   A_3225_TSC01_AT.InMonL := FALSE;
   A_3225_TSC01_AT.InMonMid := FALSE;
   A_3225_TSC01_AT.InMonH := FALSE;
   A_3225_TSC01_AT.InMonHH := FALSE;
   A_3225_TSC01_AT.spare0205 := FALSE;
   A_3225_TSC01_AT.InpFaultAI := FALSE;
   A_3225_TSC01_AT.InpFaultDev := FALSE;
   A_3225_TSC01_AT.InHWStop := FALSE;
   A_3225_TSC01_AT.InDPFault := FALSE;
   A_3225_TSC01_AT.InDisable := FALSE;
   A_3225_TSC01_AT.CmdFaultReset := FALSE;
   A_3225_TSC01_AT.InLocal := FALSE;
   A_3225_TSC01_AT.spare0305 := FALSE;
   A_3225_TSC01_AT.InReport := FALSE;
   A_3225_TSC01_AT.spare0307 := FALSE;
   A_3225_TSC01_AT.OutLL := FALSE;
   A_3225_TSC01_AT.OutL := FALSE;
   A_3225_TSC01_AT.OutH := FALSE;
   A_3225_TSC01_AT.OutHH := FALSE;
   A_3225_TSC01_AT.OutOverflow := FALSE;
   A_3225_TSC01_AT.spare0405 := FALSE;
   A_3225_TSC01_AT.OutFaultAI := FALSE;
   A_3225_TSC01_AT.spare0407 := FALSE;
   A_3225_TSC01_AT.StLL := FALSE;
   A_3225_TSC01_AT.StL := FALSE;
   A_3225_TSC01_AT.StMid := FALSE;
   A_3225_TSC01_AT.StH := FALSE;
   A_3225_TSC01_AT.StHH := FALSE;
   A_3225_TSC01_AT.StFaultAI := FALSE;
   A_3225_TSC01_AT.OutWarning := FALSE;
   A_3225_TSC01_AT.OutFaulted := FALSE;
   A_3225_TSC01_AT.InpValue := 0;
   A_3225_TSC01_AT.OutValuePc := 0;
   A_3225_TSC01_AT.OutValueUnits := L#0;
   A_3225_TSC01_AT.Msg.WarningDoneLL := FALSE;
   A_3225_TSC01_AT.Msg.WarningDoneL := FALSE;
   A_3225_TSC01_AT.Msg.WarningDoneMid := FALSE;
   A_3225_TSC01_AT.Msg.WarningDoneH := FALSE;
   A_3225_TSC01_AT.Msg.WarningDoneHH := FALSE;
   A_3225_TSC01_AT.Msg.FaultDoneLL := FALSE;
   A_3225_TSC01_AT.Msg.FaultDoneL := FALSE;
   A_3225_TSC01_AT.Msg.FaultDoneMid := FALSE;
   A_3225_TSC01_AT.Msg.FaultDoneH := FALSE;
   A_3225_TSC01_AT.Msg.FaultDoneHH := FALSE;
   A_3225_TSC01_AT.Msg.FaultDoneDev := FALSE;
   A_3225_TSC01_AT.Msg.FaultDoneAI := FALSE;
   A_3225_TSC01_AT.OutAlarmNrLog := 0;
   A_3225_TSC01_AT.Par.ParObjectNo := 29713;
   A_3225_TSC01_AT.Par.ParMsgType := 7252;
   A_3225_TSC01_AT.Par.ParHornCode := 11;
   A_3225_TSC01_AT.Par.ParLogOff := FALSE;
   A_3225_TSC01_AT.Par.ParSpare0401 := FALSE;
   A_3225_TSC01_AT.Par.ParValueByUser := FALSE;
   A_3225_TSC01_AT.Par.ParLimitsPc := TRUE;
   A_3225_TSC01_AT.Par.ParWago := FALSE;
   A_3225_TSC01_AT.Par.ParNoHornByWarning := FALSE;
   A_3225_TSC01_AT.Par.ParWarningLL := FALSE;
   A_3225_TSC01_AT.Par.ParWarningL := FALSE;
   A_3225_TSC01_AT.Par.ParWarningMid := FALSE;
   A_3225_TSC01_AT.Par.ParWarningH := FALSE;
   A_3225_TSC01_AT.Par.ParWarningHH := FALSE;
   A_3225_TSC01_AT.Par.ParPreAlarmLL := FALSE;
   A_3225_TSC01_AT.Par.ParPreAlarmL := FALSE;
   A_3225_TSC01_AT.Par.ParPreAlarmMid := FALSE;
   A_3225_TSC01_AT.Par.ParPreAlarmH := FALSE;
   A_3225_TSC01_AT.Par.ParPreAlarmHH := FALSE;
   A_3225_TSC01_AT.Par.ParUnitsByZeroDigit := L#0;
   A_3225_TSC01_AT.Par.ParUnitsByMaxDigit := L#16384;
   A_3225_TSC01_AT.Par.ParUnitsBy100Pc := L#10000;
   A_3225_TSC01_AT.Par.ParLimitLL := L#-1;
   A_3225_TSC01_AT.Par.ParLimitL := L#0;
   A_3225_TSC01_AT.Par.ParLimitH := L#7000;
   A_3225_TSC01_AT.Par.ParLimitHH := L#8000;
   A_3225_TSC01_AT.Par.ParMonTimeLL := 0;
   A_3225_TSC01_AT.Par.ParMonTimeL := 0;
   A_3225_TSC01_AT.Par.ParMonTimeMid := 0;
   A_3225_TSC01_AT.Par.ParMonTimeH := 0;
   A_3225_TSC01_AT.Par.ParMonTimeHH := 0;
   A_3225_TSC01_AT.Par.ParDelayTimeDown := 10;
   A_3225_TSC01_AT.Par.ParDelayTimeUp := 10;
   A_3225_TSC01_AT.Par.ParDelayTime := 30;
   A_3225_TSC01_AT.Par.OutMonTimeLL := 0;
   A_3225_TSC01_AT.Par.OutMonTimeL := 0;
   A_3225_TSC01_AT.Par.OutMonTimeMid := 0;
   A_3225_TSC01_AT.Par.OutMonTimeH := 0;
   A_3225_TSC01_AT.Par.OutMonTimeHH := 0;
   A_3225_TSC01_AT.Par.OutDelayTimeDown := 0;
   A_3225_TSC01_AT.Par.OutDelayTimeUp := 0;
   A_3225_TSC01_AT.Par.OutDelayTime := 0;
   A_3225_TSC01_AT.Par.Spare66 := 0;
   A_3225_TSC01_COM.InValuePC := 0;
   A_3225_TSC01_COM.InEnableRev := FALSE;
   A_3225_TSC01_COM.InEnableFwd := FALSE;
   A_3225_TSC01_COM.CmdFaultReset := FALSE;
   A_3225_TSC01_COM.OutRunningRev := FALSE;
   A_3225_TSC01_COM.OutRunningFwd := FALSE;
   A_3225_TSC01_COM.OutFault := FALSE;
   A_3225_TSC01_COM.MotorStStopped := FALSE;
   A_3225_TSC01_COM.Spare := FALSE;
   A_3225_TSC01_COM.OutValuePC := 0;
   A_3225_TSC01_COM.Input.StateWord_1.STATE_WORD_BIT_8 := FALSE;
   A_3225_TSC01_COM.Input.StateWord_1.STATE_WORD_BIT_9 := FALSE;
   A_3225_TSC01_COM.Input.StateWord_1.STATE_WORD_BIT_10 := FALSE;
   A_3225_TSC01_COM.Input.StateWord_1.STATE_WORD_BIT_11 := FALSE;
   A_3225_TSC01_COM.Input.StateWord_1.STATE_WORD_BIT_12 := FALSE;
   A_3225_TSC01_COM.Input.StateWord_1.STATE_WORD_BIT_13 := FALSE;
   A_3225_TSC01_COM.Input.StateWord_1.STATE_WORD_BIT_14 := FALSE;
   A_3225_TSC01_COM.Input.StateWord_1.STATE_WORD_BIT_15 := FALSE;
   A_3225_TSC01_COM.Input.StateWord_1.ENDSTUFE_FREIGEGEBEN := FALSE;
   A_3225_TSC01_COM.Input.StateWord_1.BETRIEBSBEREIT := FALSE;
   A_3225_TSC01_COM.Input.StateWord_1.PA_DATEN_FREIGEGEBEN := FALSE;
   A_3225_TSC01_COM.Input.StateWord_1.AKTUELL_INTEGRATORSATZ := FALSE;
   A_3225_TSC01_COM.Input.StateWord_1.AKTUELL_PARAMETERSATZ := FALSE;
   A_3225_TSC01_COM.Input.StateWord_1.STOERUNG_WARNUNG := FALSE;
   A_3225_TSC01_COM.Input.StateWord_1.LS_RECHTS_AKTIV := FALSE;
   A_3225_TSC01_COM.Input.StateWord_1.LS_LINKS_AKTIV := FALSE;
   A_3225_TSC01_COM.Input.ActualValue01 := 0;
   A_3225_TSC01_COM.Input.ActualValue02 := 0;
   A_3225_TSC01_COM.Input.ActualValue03 := 0;
   A_3225_TSC01_COM.Input.ActualValue04 := 0;
   A_3225_TSC01_COM.Input.ActualValue05 := 0;
   A_3225_TSC01_COM.Output.ControlWord_1.CONTROL_WORD_BIT_8 := FALSE;
   A_3225_TSC01_COM.Output.ControlWord_1.CONTROL_WORD_BIT_9 := FALSE;
   A_3225_TSC01_COM.Output.ControlWord_1.CONTROL_WORD_BIT_10 := FALSE;
   A_3225_TSC01_COM.Output.ControlWord_1.CONTROL_WORD_BIT_11 := FALSE;
   A_3225_TSC01_COM.Output.ControlWord_1.CONTROL_WORD_BIT_12 := FALSE;
   A_3225_TSC01_COM.Output.ControlWord_1.CONTROL_WORD_BIT_13 := FALSE;
   A_3225_TSC01_COM.Output.ControlWord_1.CONTROL_WORD_BIT_14 := FALSE;
   A_3225_TSC01_COM.Output.ControlWord_1.CONTROL_WORD_BIT_15 := FALSE;
   A_3225_TSC01_COM.Output.ControlWord_1.REGLERSPERRE := FALSE;
   A_3225_TSC01_COM.Output.ControlWord_1.FREIGABE_SCHNELLSTOPP := FALSE;
   A_3225_TSC01_COM.Output.ControlWord_1.FREIGABE_HALT := FALSE;
   A_3225_TSC01_COM.Output.ControlWord_1.HALTEREGELUNG := FALSE;
   A_3225_TSC01_COM.Output.ControlWord_1.INTEGRATOR := FALSE;
   A_3225_TSC01_COM.Output.ControlWord_1.PARAMETERSATZ := FALSE;
   A_3225_TSC01_COM.Output.ControlWord_1.RESET := FALSE;
   A_3225_TSC01_COM.Output.ControlWord_1.RESERVE_BIT_7 := FALSE;
   A_3225_TSC01_COM.Output.SetpointValue01 := 0;
   A_3225_TSC01_COM.Output.SetpointValue02 := 0;
   A_3225_TSC01_COM.Output.SetpointValue03 := 0;
   A_3225_TSC01_COM.Output.SetpointValue04 := 0;
   A_3225_TSC01_COM.Output.SetpointValue05 := 0;
   A_3225_TSC01_COM.Par.spare1 := 0;
   A_3225_TSC01_COM.Par.spare2 := 0;
   A_3225_TSC01_COM.Par.spare3 := 0;
   A_3225_TSC01_COM.Par.ParMovidrive := TRUE;
   A_3225_TSC01_COM.Par.ParSinamics := FALSE;
   A_3225_TSC01_COM.Par.ParMicromaster := FALSE;
   A_3225_TSC01_COM.Par.ParABB := FALSE;
   A_3225_TSC01_COM.Par.ParNord := FALSE;
   A_3225_TSC01_COM.Par.ParDanfoss := FALSE;
   A_3225_TSC01_COM.Par.ParIOByteNo := 0;
   A_3226_KCU04AI1.StCode := 0;
   A_3226_KCU04AI1.InMonLL := FALSE;
   A_3226_KCU04AI1.InMonL := FALSE;
   A_3226_KCU04AI1.InMonMid := FALSE;
   A_3226_KCU04AI1.InMonH := FALSE;
   A_3226_KCU04AI1.InMonHH := FALSE;
   A_3226_KCU04AI1.spare0205 := FALSE;
   A_3226_KCU04AI1.InpFaultAI := FALSE;
   A_3226_KCU04AI1.InpFaultDev := FALSE;
   A_3226_KCU04AI1.InHWStop := FALSE;
   A_3226_KCU04AI1.InDPFault := FALSE;
   A_3226_KCU04AI1.InDisable := FALSE;
   A_3226_KCU04AI1.CmdFaultReset := FALSE;
   A_3226_KCU04AI1.InLocal := FALSE;
   A_3226_KCU04AI1.spare0305 := FALSE;
   A_3226_KCU04AI1.InReport := FALSE;
   A_3226_KCU04AI1.spare0307 := FALSE;
   A_3226_KCU04AI1.OutLL := FALSE;
   A_3226_KCU04AI1.OutL := FALSE;
   A_3226_KCU04AI1.OutH := FALSE;
   A_3226_KCU04AI1.OutHH := FALSE;
   A_3226_KCU04AI1.OutOverflow := FALSE;
   A_3226_KCU04AI1.spare0405 := FALSE;
   A_3226_KCU04AI1.OutFaultAI := FALSE;
   A_3226_KCU04AI1.spare0407 := FALSE;
   A_3226_KCU04AI1.StLL := FALSE;
   A_3226_KCU04AI1.StL := FALSE;
   A_3226_KCU04AI1.StMid := FALSE;
   A_3226_KCU04AI1.StH := FALSE;
   A_3226_KCU04AI1.StHH := FALSE;
   A_3226_KCU04AI1.StFaultAI := FALSE;
   A_3226_KCU04AI1.OutWarning := FALSE;
   A_3226_KCU04AI1.OutFaulted := FALSE;
   A_3226_KCU04AI1.InpValue := 0;
   A_3226_KCU04AI1.OutValuePc := 0;
   A_3226_KCU04AI1.OutValueUnits := L#0;
   A_3226_KCU04AI1.Msg.WarningDoneLL := FALSE;
   A_3226_KCU04AI1.Msg.WarningDoneL := FALSE;
   A_3226_KCU04AI1.Msg.WarningDoneMid := FALSE;
   A_3226_KCU04AI1.Msg.WarningDoneH := FALSE;
   A_3226_KCU04AI1.Msg.WarningDoneHH := FALSE;
   A_3226_KCU04AI1.Msg.FaultDoneLL := FALSE;
   A_3226_KCU04AI1.Msg.FaultDoneL := FALSE;
   A_3226_KCU04AI1.Msg.FaultDoneMid := FALSE;
   A_3226_KCU04AI1.Msg.FaultDoneH := FALSE;
   A_3226_KCU04AI1.Msg.FaultDoneHH := FALSE;
   A_3226_KCU04AI1.Msg.FaultDoneDev := FALSE;
   A_3226_KCU04AI1.Msg.FaultDoneAI := FALSE;
   A_3226_KCU04AI1.OutAlarmNrLog := 0;
   A_3226_KCU04AI1.Par.ParObjectNo := 29715;
   A_3226_KCU04AI1.Par.ParMsgType := 7252;
   A_3226_KCU04AI1.Par.ParHornCode := 11;
   A_3226_KCU04AI1.Par.ParLogOff := FALSE;
   A_3226_KCU04AI1.Par.ParSpare0401 := FALSE;
   A_3226_KCU04AI1.Par.ParValueByUser := FALSE;
   A_3226_KCU04AI1.Par.ParLimitsPc := TRUE;
   A_3226_KCU04AI1.Par.ParWago := FALSE;
   A_3226_KCU04AI1.Par.ParNoHornByWarning := FALSE;
   A_3226_KCU04AI1.Par.ParWarningLL := FALSE;
   A_3226_KCU04AI1.Par.ParWarningL := FALSE;
   A_3226_KCU04AI1.Par.ParWarningMid := FALSE;
   A_3226_KCU04AI1.Par.ParWarningH := TRUE;
   A_3226_KCU04AI1.Par.ParWarningHH := FALSE;
   A_3226_KCU04AI1.Par.ParPreAlarmLL := FALSE;
   A_3226_KCU04AI1.Par.ParPreAlarmL := FALSE;
   A_3226_KCU04AI1.Par.ParPreAlarmMid := FALSE;
   A_3226_KCU04AI1.Par.ParPreAlarmH := FALSE;
   A_3226_KCU04AI1.Par.ParPreAlarmHH := FALSE;
   A_3226_KCU04AI1.Par.ParUnitsByZeroDigit := L#0;
   A_3226_KCU04AI1.Par.ParUnitsByMaxDigit := L#2000;
   A_3226_KCU04AI1.Par.ParUnitsBy100Pc := L#10000;
   A_3226_KCU04AI1.Par.ParLimitLL := L#-1;
   A_3226_KCU04AI1.Par.ParLimitL := L#0;
   A_3226_KCU04AI1.Par.ParLimitH := L#3150;
   A_3226_KCU04AI1.Par.ParLimitHH := L#3550;
   A_3226_KCU04AI1.Par.ParMonTimeLL := 0;
   A_3226_KCU04AI1.Par.ParMonTimeL := 0;
   A_3226_KCU04AI1.Par.ParMonTimeMid := 0;
   A_3226_KCU04AI1.Par.ParMonTimeH := 600;
   A_3226_KCU04AI1.Par.ParMonTimeHH := 0;
   A_3226_KCU04AI1.Par.ParDelayTimeDown := 10;
   A_3226_KCU04AI1.Par.ParDelayTimeUp := 10;
   A_3226_KCU04AI1.Par.ParDelayTime := 30;
   A_3226_KCU04AI1.Par.OutMonTimeLL := 0;
   A_3226_KCU04AI1.Par.OutMonTimeL := 0;
   A_3226_KCU04AI1.Par.OutMonTimeMid := 0;
   A_3226_KCU04AI1.Par.OutMonTimeH := 0;
   A_3226_KCU04AI1.Par.OutMonTimeHH := 0;
   A_3226_KCU04AI1.Par.OutDelayTimeDown := 0;
   A_3226_KCU04AI1.Par.OutDelayTimeUp := 0;
   A_3226_KCU04AI1.Par.OutDelayTime := 0;
   A_3226_KCU04AI1.Par.Spare66 := 0;
   A_3226_KCU04AI2.StCode := 0;
   A_3226_KCU04AI2.InMonLL := FALSE;
   A_3226_KCU04AI2.InMonL := FALSE;
   A_3226_KCU04AI2.InMonMid := FALSE;
   A_3226_KCU04AI2.InMonH := FALSE;
   A_3226_KCU04AI2.InMonHH := FALSE;
   A_3226_KCU04AI2.spare0205 := FALSE;
   A_3226_KCU04AI2.InpFaultAI := FALSE;
   A_3226_KCU04AI2.InpFaultDev := FALSE;
   A_3226_KCU04AI2.InHWStop := FALSE;
   A_3226_KCU04AI2.InDPFault := FALSE;
   A_3226_KCU04AI2.InDisable := FALSE;
   A_3226_KCU04AI2.CmdFaultReset := FALSE;
   A_3226_KCU04AI2.InLocal := FALSE;
   A_3226_KCU04AI2.spare0305 := FALSE;
   A_3226_KCU04AI2.InReport := FALSE;
   A_3226_KCU04AI2.spare0307 := FALSE;
   A_3226_KCU04AI2.OutLL := FALSE;
   A_3226_KCU04AI2.OutL := FALSE;
   A_3226_KCU04AI2.OutH := FALSE;
   A_3226_KCU04AI2.OutHH := FALSE;
   A_3226_KCU04AI2.OutOverflow := FALSE;
   A_3226_KCU04AI2.spare0405 := FALSE;
   A_3226_KCU04AI2.OutFaultAI := FALSE;
   A_3226_KCU04AI2.spare0407 := FALSE;
   A_3226_KCU04AI2.StLL := FALSE;
   A_3226_KCU04AI2.StL := FALSE;
   A_3226_KCU04AI2.StMid := FALSE;
   A_3226_KCU04AI2.StH := FALSE;
   A_3226_KCU04AI2.StHH := FALSE;
   A_3226_KCU04AI2.StFaultAI := FALSE;
   A_3226_KCU04AI2.OutWarning := FALSE;
   A_3226_KCU04AI2.OutFaulted := FALSE;
   A_3226_KCU04AI2.InpValue := 0;
   A_3226_KCU04AI2.OutValuePc := 0;
   A_3226_KCU04AI2.OutValueUnits := L#0;
   A_3226_KCU04AI2.Msg.WarningDoneLL := FALSE;
   A_3226_KCU04AI2.Msg.WarningDoneL := FALSE;
   A_3226_KCU04AI2.Msg.WarningDoneMid := FALSE;
   A_3226_KCU04AI2.Msg.WarningDoneH := FALSE;
   A_3226_KCU04AI2.Msg.WarningDoneHH := FALSE;
   A_3226_KCU04AI2.Msg.FaultDoneLL := FALSE;
   A_3226_KCU04AI2.Msg.FaultDoneL := FALSE;
   A_3226_KCU04AI2.Msg.FaultDoneMid := FALSE;
   A_3226_KCU04AI2.Msg.FaultDoneH := FALSE;
   A_3226_KCU04AI2.Msg.FaultDoneHH := FALSE;
   A_3226_KCU04AI2.Msg.FaultDoneDev := FALSE;
   A_3226_KCU04AI2.Msg.FaultDoneAI := FALSE;
   A_3226_KCU04AI2.OutAlarmNrLog := 0;
   A_3226_KCU04AI2.Par.ParObjectNo := 29716;
   A_3226_KCU04AI2.Par.ParMsgType := 7252;
   A_3226_KCU04AI2.Par.ParHornCode := 11;
   A_3226_KCU04AI2.Par.ParLogOff := FALSE;
   A_3226_KCU04AI2.Par.ParSpare0401 := FALSE;
   A_3226_KCU04AI2.Par.ParValueByUser := FALSE;
   A_3226_KCU04AI2.Par.ParLimitsPc := TRUE;
   A_3226_KCU04AI2.Par.ParWago := FALSE;
   A_3226_KCU04AI2.Par.ParNoHornByWarning := FALSE;
   A_3226_KCU04AI2.Par.ParWarningLL := FALSE;
   A_3226_KCU04AI2.Par.ParWarningL := FALSE;
   A_3226_KCU04AI2.Par.ParWarningMid := FALSE;
   A_3226_KCU04AI2.Par.ParWarningH := TRUE;
   A_3226_KCU04AI2.Par.ParWarningHH := FALSE;
   A_3226_KCU04AI2.Par.ParPreAlarmLL := FALSE;
   A_3226_KCU04AI2.Par.ParPreAlarmL := FALSE;
   A_3226_KCU04AI2.Par.ParPreAlarmMid := FALSE;
   A_3226_KCU04AI2.Par.ParPreAlarmH := FALSE;
   A_3226_KCU04AI2.Par.ParPreAlarmHH := FALSE;
   A_3226_KCU04AI2.Par.ParUnitsByZeroDigit := L#0;
   A_3226_KCU04AI2.Par.ParUnitsByMaxDigit := L#2000;
   A_3226_KCU04AI2.Par.ParUnitsBy100Pc := L#10000;
   A_3226_KCU04AI2.Par.ParLimitLL := L#-1;
   A_3226_KCU04AI2.Par.ParLimitL := L#0;
   A_3226_KCU04AI2.Par.ParLimitH := L#3150;
   A_3226_KCU04AI2.Par.ParLimitHH := L#3550;
   A_3226_KCU04AI2.Par.ParMonTimeLL := 0;
   A_3226_KCU04AI2.Par.ParMonTimeL := 0;
   A_3226_KCU04AI2.Par.ParMonTimeMid := 0;
   A_3226_KCU04AI2.Par.ParMonTimeH := 600;
   A_3226_KCU04AI2.Par.ParMonTimeHH := 0;
   A_3226_KCU04AI2.Par.ParDelayTimeDown := 10;
   A_3226_KCU04AI2.Par.ParDelayTimeUp := 10;
   A_3226_KCU04AI2.Par.ParDelayTime := 30;
   A_3226_KCU04AI2.Par.OutMonTimeLL := 0;
   A_3226_KCU04AI2.Par.OutMonTimeL := 0;
   A_3226_KCU04AI2.Par.OutMonTimeMid := 0;
   A_3226_KCU04AI2.Par.OutMonTimeH := 0;
   A_3226_KCU04AI2.Par.OutMonTimeHH := 0;
   A_3226_KCU04AI2.Par.OutDelayTimeDown := 0;
   A_3226_KCU04AI2.Par.OutDelayTimeUp := 0;
   A_3226_KCU04AI2.Par.OutDelayTime := 0;
   A_3226_KCU04AI2.Par.Spare66 := 0;
   A_3226_BTE05.StCode := 0;
   A_3226_BTE05.InMonLL := FALSE;
   A_3226_BTE05.InMonL := FALSE;
   A_3226_BTE05.InMonMid := FALSE;
   A_3226_BTE05.InMonH := FALSE;
   A_3226_BTE05.InMonHH := FALSE;
   A_3226_BTE05.spare0205 := FALSE;
   A_3226_BTE05.InpFaultAI := FALSE;
   A_3226_BTE05.InpFaultDev := FALSE;
   A_3226_BTE05.InHWStop := FALSE;
   A_3226_BTE05.InDPFault := FALSE;
   A_3226_BTE05.InDisable := FALSE;
   A_3226_BTE05.CmdFaultReset := FALSE;
   A_3226_BTE05.InLocal := FALSE;
   A_3226_BTE05.spare0305 := FALSE;
   A_3226_BTE05.InReport := FALSE;
   A_3226_BTE05.spare0307 := FALSE;
   A_3226_BTE05.OutLL := FALSE;
   A_3226_BTE05.OutL := FALSE;
   A_3226_BTE05.OutH := FALSE;
   A_3226_BTE05.OutHH := FALSE;
   A_3226_BTE05.OutOverflow := FALSE;
   A_3226_BTE05.spare0405 := FALSE;
   A_3226_BTE05.OutFaultAI := FALSE;
   A_3226_BTE05.spare0407 := FALSE;
   A_3226_BTE05.StLL := FALSE;
   A_3226_BTE05.StL := FALSE;
   A_3226_BTE05.StMid := FALSE;
   A_3226_BTE05.StH := FALSE;
   A_3226_BTE05.StHH := FALSE;
   A_3226_BTE05.StFaultAI := FALSE;
   A_3226_BTE05.OutWarning := FALSE;
   A_3226_BTE05.OutFaulted := FALSE;
   A_3226_BTE05.InpValue := 0;
   A_3226_BTE05.OutValuePc := 0;
   A_3226_BTE05.OutValueUnits := L#0;
   A_3226_BTE05.Msg.WarningDoneLL := FALSE;
   A_3226_BTE05.Msg.WarningDoneL := FALSE;
   A_3226_BTE05.Msg.WarningDoneMid := FALSE;
   A_3226_BTE05.Msg.WarningDoneH := FALSE;
   A_3226_BTE05.Msg.WarningDoneHH := FALSE;
   A_3226_BTE05.Msg.FaultDoneLL := FALSE;
   A_3226_BTE05.Msg.FaultDoneL := FALSE;
   A_3226_BTE05.Msg.FaultDoneMid := FALSE;
   A_3226_BTE05.Msg.FaultDoneH := FALSE;
   A_3226_BTE05.Msg.FaultDoneHH := FALSE;
   A_3226_BTE05.Msg.FaultDoneDev := FALSE;
   A_3226_BTE05.Msg.FaultDoneAI := FALSE;
   A_3226_BTE05.OutAlarmNrLog := 0;
   A_3226_BTE05.Par.ParObjectNo := 29717;
   A_3226_BTE05.Par.ParMsgType := 7252;
   A_3226_BTE05.Par.ParHornCode := 11;
   A_3226_BTE05.Par.ParLogOff := FALSE;
   A_3226_BTE05.Par.ParSpare0401 := FALSE;
   A_3226_BTE05.Par.ParValueByUser := FALSE;
   A_3226_BTE05.Par.ParLimitsPc := TRUE;
   A_3226_BTE05.Par.ParWago := FALSE;
   A_3226_BTE05.Par.ParNoHornByWarning := FALSE;
   A_3226_BTE05.Par.ParWarningLL := FALSE;
   A_3226_BTE05.Par.ParWarningL := FALSE;
   A_3226_BTE05.Par.ParWarningMid := FALSE;
   A_3226_BTE05.Par.ParWarningH := TRUE;
   A_3226_BTE05.Par.ParWarningHH := FALSE;
   A_3226_BTE05.Par.ParPreAlarmLL := FALSE;
   A_3226_BTE05.Par.ParPreAlarmL := FALSE;
   A_3226_BTE05.Par.ParPreAlarmMid := FALSE;
   A_3226_BTE05.Par.ParPreAlarmH := FALSE;
   A_3226_BTE05.Par.ParPreAlarmHH := FALSE;
   A_3226_BTE05.Par.ParUnitsByZeroDigit := L#0;
   A_3226_BTE05.Par.ParUnitsByMaxDigit := L#27384;
   A_3226_BTE05.Par.ParUnitsBy100Pc := L#10000;
   A_3226_BTE05.Par.ParLimitLL := L#0;
   A_3226_BTE05.Par.ParLimitL := L#2000;
   A_3226_BTE05.Par.ParLimitH := L#8000;
   A_3226_BTE05.Par.ParLimitHH := L#10000;
   A_3226_BTE05.Par.ParMonTimeLL := 0;
   A_3226_BTE05.Par.ParMonTimeL := 0;
   A_3226_BTE05.Par.ParMonTimeMid := 0;
   A_3226_BTE05.Par.ParMonTimeH := 600;
   A_3226_BTE05.Par.ParMonTimeHH := 0;
   A_3226_BTE05.Par.ParDelayTimeDown := 10;
   A_3226_BTE05.Par.ParDelayTimeUp := 10;
   A_3226_BTE05.Par.ParDelayTime := 30;
   A_3226_BTE05.Par.OutMonTimeLL := 0;
   A_3226_BTE05.Par.OutMonTimeL := 0;
   A_3226_BTE05.Par.OutMonTimeMid := 0;
   A_3226_BTE05.Par.OutMonTimeH := 0;
   A_3226_BTE05.Par.OutMonTimeHH := 0;
   A_3226_BTE05.Par.OutDelayTimeDown := 0;
   A_3226_BTE05.Par.OutDelayTimeUp := 0;
   A_3226_BTE05.Par.OutDelayTime := 0;
   A_3226_BTE05.Par.Spare66 := 0;
   A_3226_BTE06.StCode := 0;
   A_3226_BTE06.InMonLL := FALSE;
   A_3226_BTE06.InMonL := FALSE;
   A_3226_BTE06.InMonMid := FALSE;
   A_3226_BTE06.InMonH := FALSE;
   A_3226_BTE06.InMonHH := FALSE;
   A_3226_BTE06.spare0205 := FALSE;
   A_3226_BTE06.InpFaultAI := FALSE;
   A_3226_BTE06.InpFaultDev := FALSE;
   A_3226_BTE06.InHWStop := FALSE;
   A_3226_BTE06.InDPFault := FALSE;
   A_3226_BTE06.InDisable := FALSE;
   A_3226_BTE06.CmdFaultReset := FALSE;
   A_3226_BTE06.InLocal := FALSE;
   A_3226_BTE06.spare0305 := FALSE;
   A_3226_BTE06.InReport := FALSE;
   A_3226_BTE06.spare0307 := FALSE;
   A_3226_BTE06.OutLL := FALSE;
   A_3226_BTE06.OutL := FALSE;
   A_3226_BTE06.OutH := FALSE;
   A_3226_BTE06.OutHH := FALSE;
   A_3226_BTE06.OutOverflow := FALSE;
   A_3226_BTE06.spare0405 := FALSE;
   A_3226_BTE06.OutFaultAI := FALSE;
   A_3226_BTE06.spare0407 := FALSE;
   A_3226_BTE06.StLL := FALSE;
   A_3226_BTE06.StL := FALSE;
   A_3226_BTE06.StMid := FALSE;
   A_3226_BTE06.StH := FALSE;
   A_3226_BTE06.StHH := FALSE;
   A_3226_BTE06.StFaultAI := FALSE;
   A_3226_BTE06.OutWarning := FALSE;
   A_3226_BTE06.OutFaulted := FALSE;
   A_3226_BTE06.InpValue := 0;
   A_3226_BTE06.OutValuePc := 0;
   A_3226_BTE06.OutValueUnits := L#0;
   A_3226_BTE06.Msg.WarningDoneLL := FALSE;
   A_3226_BTE06.Msg.WarningDoneL := FALSE;
   A_3226_BTE06.Msg.WarningDoneMid := FALSE;
   A_3226_BTE06.Msg.WarningDoneH := FALSE;
   A_3226_BTE06.Msg.WarningDoneHH := FALSE;
   A_3226_BTE06.Msg.FaultDoneLL := FALSE;
   A_3226_BTE06.Msg.FaultDoneL := FALSE;
   A_3226_BTE06.Msg.FaultDoneMid := FALSE;
   A_3226_BTE06.Msg.FaultDoneH := FALSE;
   A_3226_BTE06.Msg.FaultDoneHH := FALSE;
   A_3226_BTE06.Msg.FaultDoneDev := FALSE;
   A_3226_BTE06.Msg.FaultDoneAI := FALSE;
   A_3226_BTE06.OutAlarmNrLog := 0;
   A_3226_BTE06.Par.ParObjectNo := 29718;
   A_3226_BTE06.Par.ParMsgType := 7252;
   A_3226_BTE06.Par.ParHornCode := 11;
   A_3226_BTE06.Par.ParLogOff := FALSE;
   A_3226_BTE06.Par.ParSpare0401 := FALSE;
   A_3226_BTE06.Par.ParValueByUser := FALSE;
   A_3226_BTE06.Par.ParLimitsPc := TRUE;
   A_3226_BTE06.Par.ParWago := FALSE;
   A_3226_BTE06.Par.ParNoHornByWarning := FALSE;
   A_3226_BTE06.Par.ParWarningLL := FALSE;
   A_3226_BTE06.Par.ParWarningL := FALSE;
   A_3226_BTE06.Par.ParWarningMid := FALSE;
   A_3226_BTE06.Par.ParWarningH := TRUE;
   A_3226_BTE06.Par.ParWarningHH := FALSE;
   A_3226_BTE06.Par.ParPreAlarmLL := FALSE;
   A_3226_BTE06.Par.ParPreAlarmL := FALSE;
   A_3226_BTE06.Par.ParPreAlarmMid := FALSE;
   A_3226_BTE06.Par.ParPreAlarmH := FALSE;
   A_3226_BTE06.Par.ParPreAlarmHH := FALSE;
   A_3226_BTE06.Par.ParUnitsByZeroDigit := L#0;
   A_3226_BTE06.Par.ParUnitsByMaxDigit := L#27384;
   A_3226_BTE06.Par.ParUnitsBy100Pc := L#10000;
   A_3226_BTE06.Par.ParLimitLL := L#0;
   A_3226_BTE06.Par.ParLimitL := L#2000;
   A_3226_BTE06.Par.ParLimitH := L#8000;
   A_3226_BTE06.Par.ParLimitHH := L#10000;
   A_3226_BTE06.Par.ParMonTimeLL := 0;
   A_3226_BTE06.Par.ParMonTimeL := 0;
   A_3226_BTE06.Par.ParMonTimeMid := 0;
   A_3226_BTE06.Par.ParMonTimeH := 600;
   A_3226_BTE06.Par.ParMonTimeHH := 0;
   A_3226_BTE06.Par.ParDelayTimeDown := 10;
   A_3226_BTE06.Par.ParDelayTimeUp := 10;
   A_3226_BTE06.Par.ParDelayTime := 30;
   A_3226_BTE06.Par.OutMonTimeLL := 0;
   A_3226_BTE06.Par.OutMonTimeL := 0;
   A_3226_BTE06.Par.OutMonTimeMid := 0;
   A_3226_BTE06.Par.OutMonTimeH := 0;
   A_3226_BTE06.Par.OutMonTimeHH := 0;
   A_3226_BTE06.Par.OutDelayTimeDown := 0;
   A_3226_BTE06.Par.OutDelayTimeUp := 0;
   A_3226_BTE06.Par.OutDelayTime := 0;
   A_3226_BTE06.Par.Spare66 := 0;
   A_3226_MXZ01MA.Ma.StCode := 0;
   A_3226_MXZ01MA.Ma.InEnableRev := FALSE;
   A_3226_MXZ01MA.Ma.InEnableFwd := FALSE;
   A_3226_MXZ01MA.Ma.InOverrideHLOutlet := FALSE;
   A_3226_MXZ01MA.Ma.spare0203 := FALSE;
   A_3226_MXZ01MA.Ma.OutEdgeFaultReset := FALSE;
   A_3226_MXZ01MA.Ma.OutFaultResetFcttst := FALSE;
   A_3226_MXZ01MA.Ma.InpControlEBM := FALSE;
   A_3226_MXZ01MA.Ma.InpLocked := FALSE;
   A_3226_MXZ01MA.Ma.CmdOff := FALSE;
   A_3226_MXZ01MA.Ma.CmdOn := FALSE;
   A_3226_MXZ01MA.Ma.CmdNext := FALSE;
   A_3226_MXZ01MA.Ma.CmdFaultReset := FALSE;
   A_3226_MXZ01MA.Ma.InLocal := FALSE;
   A_3226_MXZ01MA.Ma.InManual := FALSE;
   A_3226_MXZ01MA.Ma.CmdTestEBM := FALSE;
   A_3226_MXZ01MA.Ma.InSeqStop := FALSE;
   A_3226_MXZ01MA.Ma.OutWarning := FALSE;
   A_3226_MXZ01MA.Ma.InfBMTopOk := FALSE;
   A_3226_MXZ01MA.Ma.InfBMBottomOk := FALSE;
   A_3226_MXZ01MA.Ma.InfSMOk := FALSE;
   A_3226_MXZ01MA.Ma.OutpFcttst_BM_Top := FALSE;
   A_3226_MXZ01MA.Ma.OutpFcttst_BM_Bottom := FALSE;
   A_3226_MXZ01MA.Ma.OutpFcttst_SM := FALSE;
   A_3226_MXZ01MA.Ma.OutpFaultReset := FALSE;
   A_3226_MXZ01MA.Ma.StStopped := FALSE;
   A_3226_MXZ01MA.Ma.StStarting := FALSE;
   A_3226_MXZ01MA.Ma.StStartedFwd := FALSE;
   A_3226_MXZ01MA.Ma.StStopping := FALSE;
   A_3226_MXZ01MA.Ma.StFault := FALSE;
   A_3226_MXZ01MA.Ma.StStartedRev := FALSE;
   A_3226_MXZ01MA.Ma.StLocked := FALSE;
   A_3226_MXZ01MA.Ma.OutTestTime := 0;
   A_3226_MXZ01MA.Ma.Par.ParObjectNo := 29719;
   A_3226_MXZ01MA.Ma.Par.ParWithMon1 := TRUE;
   A_3226_MXZ01MA.Ma.Par.ParWithMon3 := FALSE;
   A_3226_MXZ01MA.Ma.Par.ParWithMon4 := FALSE;
   A_3226_MXZ01MA.Ma.Par.ParWithMon5 := FALSE;
   A_3226_MXZ01MA.Ma.Par.ParWithMon6 := FALSE;
   A_3226_MXZ01MA.Ma.Par.ParMon1IsHL := FALSE;
   A_3226_MXZ01MA.Ma.Par.ParMon1IsLS := TRUE;
   A_3226_MXZ01MA.Ma.Par.ParMon1StopByFault := TRUE;
   A_3226_MXZ01MA.Ma.Par.ParMon2IsLS := FALSE;
   A_3226_MXZ01MA.Ma.Par.ParMon3IsLS := FALSE;
   A_3226_MXZ01MA.Ma.Par.ParMon4AsWarning := FALSE;
   A_3226_MXZ01MA.Ma.Par.ParMon4StopByFault := FALSE;
   A_3226_MXZ01MA.Ma.Par.ParMon4IsLS := FALSE;
   A_3226_MXZ01MA.Ma.Par.ParEBM := FALSE;
   A_3226_MXZ01MA.Ma.Par.ParMon4IsSM := FALSE;
   A_3226_MXZ01MA.A_3226_KCU04.StCode := 0;
   A_3226_MXZ01MA.A_3226_KCU04.InMonTrue := FALSE;
   A_3226_MXZ01MA.A_3226_KCU04.InMonFalse := FALSE;
   A_3226_MXZ01MA.A_3226_KCU04.InPreAlarmTrue := FALSE;
   A_3226_MXZ01MA.A_3226_KCU04.InPreAlarmFalse := FALSE;
   A_3226_MXZ01MA.A_3226_KCU04.InStopTrueTime := FALSE;
   A_3226_MXZ01MA.A_3226_KCU04.InStopFalseTime := FALSE;
   A_3226_MXZ01MA.A_3226_KCU04.InpTrue := FALSE;
   A_3226_MXZ01MA.A_3226_KCU04.InpFaultDev := FALSE;
   A_3226_MXZ01MA.A_3226_KCU04.CmdRstTrueTime := FALSE;
   A_3226_MXZ01MA.A_3226_KCU04.CmdRstFalseTime := FALSE;
   A_3226_MXZ01MA.A_3226_KCU04.CmdRunTimeoutTime := FALSE;
   A_3226_MXZ01MA.A_3226_KCU04.CmdFaultReset := FALSE;
   A_3226_MXZ01MA.A_3226_KCU04.InLocal := FALSE;
   A_3226_MXZ01MA.A_3226_KCU04.spare0305 := FALSE;
   A_3226_MXZ01MA.A_3226_KCU04.InReport := FALSE;
   A_3226_MXZ01MA.A_3226_KCU04.OutTimeoutTime := FALSE;
   A_3226_MXZ01MA.A_3226_KCU04.InHWStop := FALSE;
   A_3226_MXZ01MA.A_3226_KCU04.InDPFault := FALSE;
   A_3226_MXZ01MA.A_3226_KCU04.OutPreAlarmTrue := FALSE;
   A_3226_MXZ01MA.A_3226_KCU04.OutPreAlarmFalse := FALSE;
   A_3226_MXZ01MA.A_3226_KCU04.OutFlagPos := FALSE;
   A_3226_MXZ01MA.A_3226_KCU04.OutFlagNeg := FALSE;
   A_3226_MXZ01MA.A_3226_KCU04.OutpFaultReset := FALSE;
   A_3226_MXZ01MA.A_3226_KCU04.OutTrue := FALSE;
   A_3226_MXZ01MA.A_3226_KCU04.StFalse := FALSE;
   A_3226_MXZ01MA.A_3226_KCU04.StCtoTrue := FALSE;
   A_3226_MXZ01MA.A_3226_KCU04.StTrue := FALSE;
   A_3226_MXZ01MA.A_3226_KCU04.StCtoFalse := FALSE;
   A_3226_MXZ01MA.A_3226_KCU04.StFault := FALSE;
   A_3226_MXZ01MA.A_3226_KCU04.OutAlarmNrLog := 0;
   A_3226_MXZ01MA.A_3226_KCU04.Par.ParObjectNo := 29720;
   A_3226_MXZ01MA.A_3226_KCU04.Par.ParMsgType := 7154;
   A_3226_MXZ01MA.A_3226_KCU04.Par.ParHornCode := 11;
   A_3226_MXZ01MA.A_3226_KCU04.Par.ParLogOff := FALSE;
   A_3226_MXZ01MA.A_3226_KCU04.Par.spare0401 := FALSE;
   A_3226_MXZ01MA.A_3226_KCU04.Par.Par2WorkingCond := FALSE;
   A_3226_MXZ01MA.A_3226_KCU04.Par.ParFaultRetry := FALSE;
   A_3226_MXZ01MA.A_3226_KCU04.Par.ParBinLevel := FALSE;
   A_3226_MXZ01MA.A_3226_KCU04.Par.ParDelayChange := 20;
   A_3226_MXZ01MA.A_3226_KCU04.Par.ParDelayTrue := 10;
   A_3226_MXZ01MA.A_3226_KCU04.Par.ParDelayFalse := 0;
   A_3226_MXZ01MA.A_3226_KCU04.Par.ParTimeoutTrue := 0;
   A_3226_MXZ01MA.A_3226_KCU04.Par.ParTimeoutFalse := 0;
   A_3226_MXZ01MA.A_3226_KCU04.Par.OutMonTime := 0;
   A_3226_MXZ01MA.A_3226_KCU04.Par.OutTransitionTime := 0;
   A_3226_MXZ01MA.A_3226_KCU04.Par.OutMonTrue := FALSE;
   A_3226_MXZ01MA.A_3226_KCU04.Par.OutMonFalse := FALSE;
   A_3226_MXZ01MA.A_3226_KCU04.Par.OutFlagFaultDev := FALSE;
   A_3226_MXZ01MA.A_3226_KCU04.Par.OutDelayTime := 0;
   A_3226_MXZ01MA.A_3226_MXZ01_SM.StCode := 0;
   A_3226_MXZ01MA.A_3226_MXZ01_SM.InMonTrue := FALSE;
   A_3226_MXZ01MA.A_3226_MXZ01_SM.InMonFalse := FALSE;
   A_3226_MXZ01MA.A_3226_MXZ01_SM.InPreAlarmTrue := FALSE;
   A_3226_MXZ01MA.A_3226_MXZ01_SM.InPreAlarmFalse := FALSE;
   A_3226_MXZ01MA.A_3226_MXZ01_SM.InStopTrueTime := FALSE;
   A_3226_MXZ01MA.A_3226_MXZ01_SM.InStopFalseTime := FALSE;
   A_3226_MXZ01MA.A_3226_MXZ01_SM.InpTrue := FALSE;
   A_3226_MXZ01MA.A_3226_MXZ01_SM.InpFaultDev := FALSE;
   A_3226_MXZ01MA.A_3226_MXZ01_SM.CmdRstTrueTime := FALSE;
   A_3226_MXZ01MA.A_3226_MXZ01_SM.CmdRstFalseTime := FALSE;
   A_3226_MXZ01MA.A_3226_MXZ01_SM.CmdRunTimeoutTime := FALSE;
   A_3226_MXZ01MA.A_3226_MXZ01_SM.CmdFaultReset := FALSE;
   A_3226_MXZ01MA.A_3226_MXZ01_SM.InLocal := FALSE;
   A_3226_MXZ01MA.A_3226_MXZ01_SM.spare0305 := FALSE;
   A_3226_MXZ01MA.A_3226_MXZ01_SM.InReport := FALSE;
   A_3226_MXZ01MA.A_3226_MXZ01_SM.OutTimeoutTime := FALSE;
   A_3226_MXZ01MA.A_3226_MXZ01_SM.InHWStop := FALSE;
   A_3226_MXZ01MA.A_3226_MXZ01_SM.InDPFault := FALSE;
   A_3226_MXZ01MA.A_3226_MXZ01_SM.OutPreAlarmTrue := FALSE;
   A_3226_MXZ01MA.A_3226_MXZ01_SM.OutPreAlarmFalse := FALSE;
   A_3226_MXZ01MA.A_3226_MXZ01_SM.OutFlagPos := FALSE;
   A_3226_MXZ01MA.A_3226_MXZ01_SM.OutFlagNeg := FALSE;
   A_3226_MXZ01MA.A_3226_MXZ01_SM.OutpFaultReset := FALSE;
   A_3226_MXZ01MA.A_3226_MXZ01_SM.OutTrue := FALSE;
   A_3226_MXZ01MA.A_3226_MXZ01_SM.StFalse := FALSE;
   A_3226_MXZ01MA.A_3226_MXZ01_SM.StCtoTrue := FALSE;
   A_3226_MXZ01MA.A_3226_MXZ01_SM.StTrue := FALSE;
   A_3226_MXZ01MA.A_3226_MXZ01_SM.StCtoFalse := FALSE;
   A_3226_MXZ01MA.A_3226_MXZ01_SM.StFault := FALSE;
   A_3226_MXZ01MA.A_3226_MXZ01_SM.OutAlarmNrLog := 0;
   A_3226_MXZ01MA.A_3226_MXZ01_SM.Par.ParObjectNo := 29721;
   A_3226_MXZ01MA.A_3226_MXZ01_SM.Par.ParMsgType := 7135;
   A_3226_MXZ01MA.A_3226_MXZ01_SM.Par.ParHornCode := 11;
   A_3226_MXZ01MA.A_3226_MXZ01_SM.Par.ParLogOff := FALSE;
   A_3226_MXZ01MA.A_3226_MXZ01_SM.Par.spare0401 := FALSE;
   A_3226_MXZ01MA.A_3226_MXZ01_SM.Par.Par2WorkingCond := TRUE;
   A_3226_MXZ01MA.A_3226_MXZ01_SM.Par.ParFaultRetry := FALSE;
   A_3226_MXZ01MA.A_3226_MXZ01_SM.Par.ParBinLevel := FALSE;
   A_3226_MXZ01MA.A_3226_MXZ01_SM.Par.ParDelayChange := 0;
   A_3226_MXZ01MA.A_3226_MXZ01_SM.Par.ParDelayTrue := 10;
   A_3226_MXZ01MA.A_3226_MXZ01_SM.Par.ParDelayFalse := 0;
   A_3226_MXZ01MA.A_3226_MXZ01_SM.Par.ParTimeoutTrue := 50;
   A_3226_MXZ01MA.A_3226_MXZ01_SM.Par.ParTimeoutFalse := 0;
   A_3226_MXZ01MA.A_3226_MXZ01_SM.Par.OutMonTime := 0;
   A_3226_MXZ01MA.A_3226_MXZ01_SM.Par.OutTransitionTime := 0;
   A_3226_MXZ01MA.A_3226_MXZ01_SM.Par.OutMonTrue := FALSE;
   A_3226_MXZ01MA.A_3226_MXZ01_SM.Par.OutMonFalse := FALSE;
   A_3226_MXZ01MA.A_3226_MXZ01_SM.Par.OutFlagFaultDev := FALSE;
   A_3226_MXZ01MA.A_3226_MXZ01_SM.Par.OutDelayTime := 0;
   A_3226_MXZ01MA.Mon3.StCode := 0;
   A_3226_MXZ01MA.Mon3.InMonTrue := FALSE;
   A_3226_MXZ01MA.Mon3.InMonFalse := FALSE;
   A_3226_MXZ01MA.Mon3.InPreAlarmTrue := FALSE;
   A_3226_MXZ01MA.Mon3.InPreAlarmFalse := FALSE;
   A_3226_MXZ01MA.Mon3.InStopTrueTime := FALSE;
   A_3226_MXZ01MA.Mon3.InStopFalseTime := FALSE;
   A_3226_MXZ01MA.Mon3.InpTrue := FALSE;
   A_3226_MXZ01MA.Mon3.InpFaultDev := FALSE;
   A_3226_MXZ01MA.Mon3.CmdRstTrueTime := FALSE;
   A_3226_MXZ01MA.Mon3.CmdRstFalseTime := FALSE;
   A_3226_MXZ01MA.Mon3.CmdRunTimeoutTime := FALSE;
   A_3226_MXZ01MA.Mon3.CmdFaultReset := FALSE;
   A_3226_MXZ01MA.Mon3.InLocal := FALSE;
   A_3226_MXZ01MA.Mon3.spare0305 := FALSE;
   A_3226_MXZ01MA.Mon3.InReport := FALSE;
   A_3226_MXZ01MA.Mon3.OutTimeoutTime := FALSE;
   A_3226_MXZ01MA.Mon3.InHWStop := FALSE;
   A_3226_MXZ01MA.Mon3.InDPFault := FALSE;
   A_3226_MXZ01MA.Mon3.OutPreAlarmTrue := FALSE;
   A_3226_MXZ01MA.Mon3.OutPreAlarmFalse := FALSE;
   A_3226_MXZ01MA.Mon3.OutFlagPos := FALSE;
   A_3226_MXZ01MA.Mon3.OutFlagNeg := FALSE;
   A_3226_MXZ01MA.Mon3.OutpFaultReset := FALSE;
   A_3226_MXZ01MA.Mon3.OutTrue := FALSE;
   A_3226_MXZ01MA.Mon3.StFalse := FALSE;
   A_3226_MXZ01MA.Mon3.StCtoTrue := FALSE;
   A_3226_MXZ01MA.Mon3.StTrue := FALSE;
   A_3226_MXZ01MA.Mon3.StCtoFalse := FALSE;
   A_3226_MXZ01MA.Mon3.StFault := FALSE;
   A_3226_MXZ01MA.Mon3.OutAlarmNrLog := 0;
   A_3226_MXZ01MA.Mon3.Par.ParObjectNo := 0;
   A_3226_MXZ01MA.Mon3.Par.ParMsgType := 0;
   A_3226_MXZ01MA.Mon3.Par.ParHornCode := 0;
   A_3226_MXZ01MA.Mon3.Par.ParLogOff := FALSE;
   A_3226_MXZ01MA.Mon3.Par.spare0401 := FALSE;
   A_3226_MXZ01MA.Mon3.Par.Par2WorkingCond := FALSE;
   A_3226_MXZ01MA.Mon3.Par.ParFaultRetry := FALSE;
   A_3226_MXZ01MA.Mon3.Par.ParBinLevel := FALSE;
   A_3226_MXZ01MA.Mon3.Par.ParDelayChange := 0;
   A_3226_MXZ01MA.Mon3.Par.ParDelayTrue := 0;
   A_3226_MXZ01MA.Mon3.Par.ParDelayFalse := 0;
   A_3226_MXZ01MA.Mon3.Par.ParTimeoutTrue := 0;
   A_3226_MXZ01MA.Mon3.Par.ParTimeoutFalse := 0;
   A_3226_MXZ01MA.Mon3.Par.OutMonTime := 0;
   A_3226_MXZ01MA.Mon3.Par.OutTransitionTime := 0;
   A_3226_MXZ01MA.Mon3.Par.OutMonTrue := FALSE;
   A_3226_MXZ01MA.Mon3.Par.OutMonFalse := FALSE;
   A_3226_MXZ01MA.Mon3.Par.OutFlagFaultDev := FALSE;
   A_3226_MXZ01MA.Mon3.Par.OutDelayTime := 0;
   A_3226_MXZ01MA.Mon4.StCode := 0;
   A_3226_MXZ01MA.Mon4.InMonTrue := FALSE;
   A_3226_MXZ01MA.Mon4.InMonFalse := FALSE;
   A_3226_MXZ01MA.Mon4.InPreAlarmTrue := FALSE;
   A_3226_MXZ01MA.Mon4.InPreAlarmFalse := FALSE;
   A_3226_MXZ01MA.Mon4.InStopTrueTime := FALSE;
   A_3226_MXZ01MA.Mon4.InStopFalseTime := FALSE;
   A_3226_MXZ01MA.Mon4.InpTrue := FALSE;
   A_3226_MXZ01MA.Mon4.InpFaultDev := FALSE;
   A_3226_MXZ01MA.Mon4.CmdRstTrueTime := FALSE;
   A_3226_MXZ01MA.Mon4.CmdRstFalseTime := FALSE;
   A_3226_MXZ01MA.Mon4.CmdRunTimeoutTime := FALSE;
   A_3226_MXZ01MA.Mon4.CmdFaultReset := FALSE;
   A_3226_MXZ01MA.Mon4.InLocal := FALSE;
   A_3226_MXZ01MA.Mon4.spare0305 := FALSE;
   A_3226_MXZ01MA.Mon4.InReport := FALSE;
   A_3226_MXZ01MA.Mon4.OutTimeoutTime := FALSE;
   A_3226_MXZ01MA.Mon4.InHWStop := FALSE;
   A_3226_MXZ01MA.Mon4.InDPFault := FALSE;
   A_3226_MXZ01MA.Mon4.OutPreAlarmTrue := FALSE;
   A_3226_MXZ01MA.Mon4.OutPreAlarmFalse := FALSE;
   A_3226_MXZ01MA.Mon4.OutFlagPos := FALSE;
   A_3226_MXZ01MA.Mon4.OutFlagNeg := FALSE;
   A_3226_MXZ01MA.Mon4.OutpFaultReset := FALSE;
   A_3226_MXZ01MA.Mon4.OutTrue := FALSE;
   A_3226_MXZ01MA.Mon4.StFalse := FALSE;
   A_3226_MXZ01MA.Mon4.StCtoTrue := FALSE;
   A_3226_MXZ01MA.Mon4.StTrue := FALSE;
   A_3226_MXZ01MA.Mon4.StCtoFalse := FALSE;
   A_3226_MXZ01MA.Mon4.StFault := FALSE;
   A_3226_MXZ01MA.Mon4.OutAlarmNrLog := 0;
   A_3226_MXZ01MA.Mon4.Par.ParObjectNo := 0;
   A_3226_MXZ01MA.Mon4.Par.ParMsgType := 0;
   A_3226_MXZ01MA.Mon4.Par.ParHornCode := 0;
   A_3226_MXZ01MA.Mon4.Par.ParLogOff := FALSE;
   A_3226_MXZ01MA.Mon4.Par.spare0401 := FALSE;
   A_3226_MXZ01MA.Mon4.Par.Par2WorkingCond := FALSE;
   A_3226_MXZ01MA.Mon4.Par.ParFaultRetry := FALSE;
   A_3226_MXZ01MA.Mon4.Par.ParBinLevel := FALSE;
   A_3226_MXZ01MA.Mon4.Par.ParDelayChange := 0;
   A_3226_MXZ01MA.Mon4.Par.ParDelayTrue := 0;
   A_3226_MXZ01MA.Mon4.Par.ParDelayFalse := 0;
   A_3226_MXZ01MA.Mon4.Par.ParTimeoutTrue := 0;
   A_3226_MXZ01MA.Mon4.Par.ParTimeoutFalse := 0;
   A_3226_MXZ01MA.Mon4.Par.OutMonTime := 0;
   A_3226_MXZ01MA.Mon4.Par.OutTransitionTime := 0;
   A_3226_MXZ01MA.Mon4.Par.OutMonTrue := FALSE;
   A_3226_MXZ01MA.Mon4.Par.OutMonFalse := FALSE;
   A_3226_MXZ01MA.Mon4.Par.OutFlagFaultDev := FALSE;
   A_3226_MXZ01MA.Mon4.Par.OutDelayTime := 0;
   A_3226_MXZ01MA.Mon5.StCode := 0;
   A_3226_MXZ01MA.Mon5.InMonTrue := FALSE;
   A_3226_MXZ01MA.Mon5.InMonFalse := FALSE;
   A_3226_MXZ01MA.Mon5.InPreAlarmTrue := FALSE;
   A_3226_MXZ01MA.Mon5.InPreAlarmFalse := FALSE;
   A_3226_MXZ01MA.Mon5.InStopTrueTime := FALSE;
   A_3226_MXZ01MA.Mon5.InStopFalseTime := FALSE;
   A_3226_MXZ01MA.Mon5.InpTrue := FALSE;
   A_3226_MXZ01MA.Mon5.InpFaultDev := FALSE;
   A_3226_MXZ01MA.Mon5.CmdRstTrueTime := FALSE;
   A_3226_MXZ01MA.Mon5.CmdRstFalseTime := FALSE;
   A_3226_MXZ01MA.Mon5.CmdRunTimeoutTime := FALSE;
   A_3226_MXZ01MA.Mon5.CmdFaultReset := FALSE;
   A_3226_MXZ01MA.Mon5.InLocal := FALSE;
   A_3226_MXZ01MA.Mon5.spare0305 := FALSE;
   A_3226_MXZ01MA.Mon5.InReport := FALSE;
   A_3226_MXZ01MA.Mon5.OutTimeoutTime := FALSE;
   A_3226_MXZ01MA.Mon5.InHWStop := FALSE;
   A_3226_MXZ01MA.Mon5.InDPFault := FALSE;
   A_3226_MXZ01MA.Mon5.OutPreAlarmTrue := FALSE;
   A_3226_MXZ01MA.Mon5.OutPreAlarmFalse := FALSE;
   A_3226_MXZ01MA.Mon5.OutFlagPos := FALSE;
   A_3226_MXZ01MA.Mon5.OutFlagNeg := FALSE;
   A_3226_MXZ01MA.Mon5.OutpFaultReset := FALSE;
   A_3226_MXZ01MA.Mon5.OutTrue := FALSE;
   A_3226_MXZ01MA.Mon5.StFalse := FALSE;
   A_3226_MXZ01MA.Mon5.StCtoTrue := FALSE;
   A_3226_MXZ01MA.Mon5.StTrue := FALSE;
   A_3226_MXZ01MA.Mon5.StCtoFalse := FALSE;
   A_3226_MXZ01MA.Mon5.StFault := FALSE;
   A_3226_MXZ01MA.Mon5.OutAlarmNrLog := 0;
   A_3226_MXZ01MA.Mon5.Par.ParObjectNo := 0;
   A_3226_MXZ01MA.Mon5.Par.ParMsgType := 0;
   A_3226_MXZ01MA.Mon5.Par.ParHornCode := 0;
   A_3226_MXZ01MA.Mon5.Par.ParLogOff := FALSE;
   A_3226_MXZ01MA.Mon5.Par.spare0401 := FALSE;
   A_3226_MXZ01MA.Mon5.Par.Par2WorkingCond := FALSE;
   A_3226_MXZ01MA.Mon5.Par.ParFaultRetry := FALSE;
   A_3226_MXZ01MA.Mon5.Par.ParBinLevel := FALSE;
   A_3226_MXZ01MA.Mon5.Par.ParDelayChange := 0;
   A_3226_MXZ01MA.Mon5.Par.ParDelayTrue := 0;
   A_3226_MXZ01MA.Mon5.Par.ParDelayFalse := 0;
   A_3226_MXZ01MA.Mon5.Par.ParTimeoutTrue := 0;
   A_3226_MXZ01MA.Mon5.Par.ParTimeoutFalse := 0;
   A_3226_MXZ01MA.Mon5.Par.OutMonTime := 0;
   A_3226_MXZ01MA.Mon5.Par.OutTransitionTime := 0;
   A_3226_MXZ01MA.Mon5.Par.OutMonTrue := FALSE;
   A_3226_MXZ01MA.Mon5.Par.OutMonFalse := FALSE;
   A_3226_MXZ01MA.Mon5.Par.OutFlagFaultDev := FALSE;
   A_3226_MXZ01MA.Mon5.Par.OutDelayTime := 0;
   A_3226_MXZ01MA.Mon6.StCode := 0;
   A_3226_MXZ01MA.Mon6.InMonTrue := FALSE;
   A_3226_MXZ01MA.Mon6.InMonFalse := FALSE;
   A_3226_MXZ01MA.Mon6.InPreAlarmTrue := FALSE;
   A_3226_MXZ01MA.Mon6.InPreAlarmFalse := FALSE;
   A_3226_MXZ01MA.Mon6.InStopTrueTime := FALSE;
   A_3226_MXZ01MA.Mon6.InStopFalseTime := FALSE;
   A_3226_MXZ01MA.Mon6.InpTrue := FALSE;
   A_3226_MXZ01MA.Mon6.InpFaultDev := FALSE;
   A_3226_MXZ01MA.Mon6.CmdRstTrueTime := FALSE;
   A_3226_MXZ01MA.Mon6.CmdRstFalseTime := FALSE;
   A_3226_MXZ01MA.Mon6.CmdRunTimeoutTime := FALSE;
   A_3226_MXZ01MA.Mon6.CmdFaultReset := FALSE;
   A_3226_MXZ01MA.Mon6.InLocal := FALSE;
   A_3226_MXZ01MA.Mon6.spare0305 := FALSE;
   A_3226_MXZ01MA.Mon6.InReport := FALSE;
   A_3226_MXZ01MA.Mon6.OutTimeoutTime := FALSE;
   A_3226_MXZ01MA.Mon6.InHWStop := FALSE;
   A_3226_MXZ01MA.Mon6.InDPFault := FALSE;
   A_3226_MXZ01MA.Mon6.OutPreAlarmTrue := FALSE;
   A_3226_MXZ01MA.Mon6.OutPreAlarmFalse := FALSE;
   A_3226_MXZ01MA.Mon6.OutFlagPos := FALSE;
   A_3226_MXZ01MA.Mon6.OutFlagNeg := FALSE;
   A_3226_MXZ01MA.Mon6.OutpFaultReset := FALSE;
   A_3226_MXZ01MA.Mon6.OutTrue := FALSE;
   A_3226_MXZ01MA.Mon6.StFalse := FALSE;
   A_3226_MXZ01MA.Mon6.StCtoTrue := FALSE;
   A_3226_MXZ01MA.Mon6.StTrue := FALSE;
   A_3226_MXZ01MA.Mon6.StCtoFalse := FALSE;
   A_3226_MXZ01MA.Mon6.StFault := FALSE;
   A_3226_MXZ01MA.Mon6.OutAlarmNrLog := 0;
   A_3226_MXZ01MA.Mon6.Par.ParObjectNo := 0;
   A_3226_MXZ01MA.Mon6.Par.ParMsgType := 0;
   A_3226_MXZ01MA.Mon6.Par.ParHornCode := 0;
   A_3226_MXZ01MA.Mon6.Par.ParLogOff := FALSE;
   A_3226_MXZ01MA.Mon6.Par.spare0401 := FALSE;
   A_3226_MXZ01MA.Mon6.Par.Par2WorkingCond := FALSE;
   A_3226_MXZ01MA.Mon6.Par.ParFaultRetry := FALSE;
   A_3226_MXZ01MA.Mon6.Par.ParBinLevel := FALSE;
   A_3226_MXZ01MA.Mon6.Par.ParDelayChange := 0;
   A_3226_MXZ01MA.Mon6.Par.ParDelayTrue := 0;
   A_3226_MXZ01MA.Mon6.Par.ParDelayFalse := 0;
   A_3226_MXZ01MA.Mon6.Par.ParTimeoutTrue := 0;
   A_3226_MXZ01MA.Mon6.Par.ParTimeoutFalse := 0;
   A_3226_MXZ01MA.Mon6.Par.OutMonTime := 0;
   A_3226_MXZ01MA.Mon6.Par.OutTransitionTime := 0;
   A_3226_MXZ01MA.Mon6.Par.OutMonTrue := FALSE;
   A_3226_MXZ01MA.Mon6.Par.OutMonFalse := FALSE;
   A_3226_MXZ01MA.Mon6.Par.OutFlagFaultDev := FALSE;
   A_3226_MXZ01MA.Mon6.Par.OutDelayTime := 0;
   A_3226_MXZ01MA.A_3226_MXZ01.StCode := 0;
   A_3226_MXZ01MA.A_3226_MXZ01.InEnableRev := FALSE;
   A_3226_MXZ01MA.A_3226_MXZ01.InEnableFwd := FALSE;
   A_3226_MXZ01MA.A_3226_MXZ01.InSlow := FALSE;
   A_3226_MXZ01MA.A_3226_MXZ01.InpRunSlow := FALSE;
   A_3226_MXZ01MA.A_3226_MXZ01.InpRunFast := FALSE;
   A_3226_MXZ01MA.A_3226_MXZ01.InpRunRev := FALSE;
   A_3226_MXZ01MA.A_3226_MXZ01.InpRunFwd := FALSE;
   A_3226_MXZ01MA.A_3226_MXZ01.InpFaultDev := FALSE;
   A_3226_MXZ01MA.A_3226_MXZ01.CmdOff := FALSE;
   A_3226_MXZ01MA.A_3226_MXZ01.CmdOn := FALSE;
   A_3226_MXZ01MA.A_3226_MXZ01.CmdNext := FALSE;
   A_3226_MXZ01MA.A_3226_MXZ01.CmdFaultReset := FALSE;
   A_3226_MXZ01MA.A_3226_MXZ01.InLocal := FALSE;
   A_3226_MXZ01MA.A_3226_MXZ01.InManual := FALSE;
   A_3226_MXZ01MA.A_3226_MXZ01.InReport := FALSE;
   A_3226_MXZ01MA.A_3226_MXZ01.InSeqStop := FALSE;
   A_3226_MXZ01MA.A_3226_MXZ01.InHWStop := FALSE;
   A_3226_MXZ01MA.A_3226_MXZ01.InDPFault := FALSE;
   A_3226_MXZ01MA.A_3226_MXZ01.OutIdling := FALSE;
   A_3226_MXZ01MA.A_3226_MXZ01.OutpRunSlow := FALSE;
   A_3226_MXZ01MA.A_3226_MXZ01.OutpRunFast := FALSE;
   A_3226_MXZ01MA.A_3226_MXZ01.OutpRunRev := FALSE;
   A_3226_MXZ01MA.A_3226_MXZ01.OutpRunFwd := FALSE;
   A_3226_MXZ01MA.A_3226_MXZ01.OutpFaultReset := FALSE;
   A_3226_MXZ01MA.A_3226_MXZ01.StStopped := FALSE;
   A_3226_MXZ01MA.A_3226_MXZ01.StStarting := FALSE;
   A_3226_MXZ01MA.A_3226_MXZ01.StStartedFwd := FALSE;
   A_3226_MXZ01MA.A_3226_MXZ01.StStopping := FALSE;
   A_3226_MXZ01MA.A_3226_MXZ01.StFault := FALSE;
   A_3226_MXZ01MA.A_3226_MXZ01.StStartedRev := FALSE;
   A_3226_MXZ01MA.A_3226_MXZ01.InOutManSlow := FALSE;
   A_3226_MXZ01MA.A_3226_MXZ01.InOutManRev := FALSE;
   A_3226_MXZ01MA.A_3226_MXZ01.OutAlarmNrLog := 0;
   A_3226_MXZ01MA.A_3226_MXZ01.Par.ParObjectNo := 29722;
   A_3226_MXZ01MA.A_3226_MXZ01.Par.ParMsgType := 7053;
   A_3226_MXZ01MA.A_3226_MXZ01.Par.ParHornCode := 11;
   A_3226_MXZ01MA.A_3226_MXZ01.Par.ParLogOff := FALSE;
   A_3226_MXZ01MA.A_3226_MXZ01.Par.ParManual := TRUE;
   A_3226_MXZ01MA.A_3226_MXZ01.Par.ParRestartDelay := FALSE;
   A_3226_MXZ01MA.A_3226_MXZ01.Par.Par2Speed := FALSE;
   A_3226_MXZ01MA.A_3226_MXZ01.Par.ParHeavyStartup := FALSE;
   A_3226_MXZ01MA.A_3226_MXZ01.Par.spare45 := FALSE;
   A_3226_MXZ01MA.A_3226_MXZ01.Par.spare46 := FALSE;
   A_3226_MXZ01MA.A_3226_MXZ01.Par.OutEdgeFaultReset := FALSE;
   A_3226_MXZ01MA.A_3226_MXZ01.Par.OutDelayFault := FALSE;
   A_3226_MXZ01MA.A_3226_MXZ01.Par.OutFlagFaultDev := FALSE;
   A_3226_MXZ01MA.A_3226_MXZ01.Par.ParMonTime := 20;
   A_3226_MXZ01MA.A_3226_MXZ01.Par.ParStartingTime := 20;
   A_3226_MXZ01MA.A_3226_MXZ01.Par.ParStoppingTime := 0;
   A_3226_MXZ01MA.A_3226_MXZ01.Par.ParIdlingTime := 0;
   A_3226_MXZ01MA.A_3226_MXZ01.Par.ParDelayTime := 10;
   A_3226_MXZ01MA.A_3226_MXZ01.Par.OutMonTime := 0;
   A_3226_MXZ01MA.A_3226_MXZ01.Par.OutTransitionTime := 0;
   A_3226_MXZ01MA.A_3226_MXZ01.Par.OutDelayTime := 0;
   A_3226_MXZ01MA.A_3226_MXZ01.Par.InOutManPulseLen := 0;
   A_3226_TSC01_AC.StCode := 0;
   A_3226_TSC01_AC.InMonLL := FALSE;
   A_3226_TSC01_AC.InMonL := FALSE;
   A_3226_TSC01_AC.InMonMid := FALSE;
   A_3226_TSC01_AC.InMonH := FALSE;
   A_3226_TSC01_AC.InMonHH := FALSE;
   A_3226_TSC01_AC.spare0205 := FALSE;
   A_3226_TSC01_AC.InpFaultAI := FALSE;
   A_3226_TSC01_AC.InpFaultDev := FALSE;
   A_3226_TSC01_AC.InHWStop := FALSE;
   A_3226_TSC01_AC.InDPFault := FALSE;
   A_3226_TSC01_AC.InDisable := FALSE;
   A_3226_TSC01_AC.CmdFaultReset := FALSE;
   A_3226_TSC01_AC.InLocal := FALSE;
   A_3226_TSC01_AC.spare0305 := FALSE;
   A_3226_TSC01_AC.InReport := FALSE;
   A_3226_TSC01_AC.spare0307 := FALSE;
   A_3226_TSC01_AC.OutLL := FALSE;
   A_3226_TSC01_AC.OutL := FALSE;
   A_3226_TSC01_AC.OutH := FALSE;
   A_3226_TSC01_AC.OutHH := FALSE;
   A_3226_TSC01_AC.OutOverflow := FALSE;
   A_3226_TSC01_AC.spare0405 := FALSE;
   A_3226_TSC01_AC.OutFaultAI := FALSE;
   A_3226_TSC01_AC.spare0407 := FALSE;
   A_3226_TSC01_AC.StLL := FALSE;
   A_3226_TSC01_AC.StL := FALSE;
   A_3226_TSC01_AC.StMid := FALSE;
   A_3226_TSC01_AC.StH := FALSE;
   A_3226_TSC01_AC.StHH := FALSE;
   A_3226_TSC01_AC.StFaultAI := FALSE;
   A_3226_TSC01_AC.OutWarning := FALSE;
   A_3226_TSC01_AC.OutFaulted := FALSE;
   A_3226_TSC01_AC.InpValue := 0;
   A_3226_TSC01_AC.OutValuePc := 0;
   A_3226_TSC01_AC.OutValueUnits := L#0;
   A_3226_TSC01_AC.Msg.WarningDoneLL := FALSE;
   A_3226_TSC01_AC.Msg.WarningDoneL := FALSE;
   A_3226_TSC01_AC.Msg.WarningDoneMid := FALSE;
   A_3226_TSC01_AC.Msg.WarningDoneH := FALSE;
   A_3226_TSC01_AC.Msg.WarningDoneHH := FALSE;
   A_3226_TSC01_AC.Msg.FaultDoneLL := FALSE;
   A_3226_TSC01_AC.Msg.FaultDoneL := FALSE;
   A_3226_TSC01_AC.Msg.FaultDoneMid := FALSE;
   A_3226_TSC01_AC.Msg.FaultDoneH := FALSE;
   A_3226_TSC01_AC.Msg.FaultDoneHH := FALSE;
   A_3226_TSC01_AC.Msg.FaultDoneDev := FALSE;
   A_3226_TSC01_AC.Msg.FaultDoneAI := FALSE;
   A_3226_TSC01_AC.OutAlarmNrLog := 0;
   A_3226_TSC01_AC.Par.ParObjectNo := 29723;
   A_3226_TSC01_AC.Par.ParMsgType := 7252;
   A_3226_TSC01_AC.Par.ParHornCode := 11;
   A_3226_TSC01_AC.Par.ParLogOff := FALSE;
   A_3226_TSC01_AC.Par.ParSpare0401 := FALSE;
   A_3226_TSC01_AC.Par.ParValueByUser := FALSE;
   A_3226_TSC01_AC.Par.ParLimitsPc := TRUE;
   A_3226_TSC01_AC.Par.ParWago := FALSE;
   A_3226_TSC01_AC.Par.ParNoHornByWarning := FALSE;
   A_3226_TSC01_AC.Par.ParWarningLL := FALSE;
   A_3226_TSC01_AC.Par.ParWarningL := FALSE;
   A_3226_TSC01_AC.Par.ParWarningMid := FALSE;
   A_3226_TSC01_AC.Par.ParWarningH := FALSE;
   A_3226_TSC01_AC.Par.ParWarningHH := FALSE;
   A_3226_TSC01_AC.Par.ParPreAlarmLL := FALSE;
   A_3226_TSC01_AC.Par.ParPreAlarmL := FALSE;
   A_3226_TSC01_AC.Par.ParPreAlarmMid := FALSE;
   A_3226_TSC01_AC.Par.ParPreAlarmH := FALSE;
   A_3226_TSC01_AC.Par.ParPreAlarmHH := FALSE;
   A_3226_TSC01_AC.Par.ParUnitsByZeroDigit := L#0;
   A_3226_TSC01_AC.Par.ParUnitsByMaxDigit := L#25384;
   A_3226_TSC01_AC.Par.ParUnitsBy100Pc := L#10000;
   A_3226_TSC01_AC.Par.ParLimitLL := L#-1;
   A_3226_TSC01_AC.Par.ParLimitL := L#0;
   A_3226_TSC01_AC.Par.ParLimitH := L#5400;
   A_3226_TSC01_AC.Par.ParLimitHH := L#6000;
   A_3226_TSC01_AC.Par.ParMonTimeLL := 0;
   A_3226_TSC01_AC.Par.ParMonTimeL := 0;
   A_3226_TSC01_AC.Par.ParMonTimeMid := 0;
   A_3226_TSC01_AC.Par.ParMonTimeH := 0;
   A_3226_TSC01_AC.Par.ParMonTimeHH := 0;
   A_3226_TSC01_AC.Par.ParDelayTimeDown := 10;
   A_3226_TSC01_AC.Par.ParDelayTimeUp := 10;
   A_3226_TSC01_AC.Par.ParDelayTime := 30;
   A_3226_TSC01_AC.Par.OutMonTimeLL := 0;
   A_3226_TSC01_AC.Par.OutMonTimeL := 0;
   A_3226_TSC01_AC.Par.OutMonTimeMid := 0;
   A_3226_TSC01_AC.Par.OutMonTimeH := 0;
   A_3226_TSC01_AC.Par.OutMonTimeHH := 0;
   A_3226_TSC01_AC.Par.OutDelayTimeDown := 0;
   A_3226_TSC01_AC.Par.OutDelayTimeUp := 0;
   A_3226_TSC01_AC.Par.OutDelayTime := 0;
   A_3226_TSC01_AC.Par.Spare66 := 0;
   A_3226_TSC01_AF.StCode := 0;
   A_3226_TSC01_AF.InMonLL := FALSE;
   A_3226_TSC01_AF.InMonL := FALSE;
   A_3226_TSC01_AF.InMonMid := FALSE;
   A_3226_TSC01_AF.InMonH := FALSE;
   A_3226_TSC01_AF.InMonHH := FALSE;
   A_3226_TSC01_AF.spare0205 := FALSE;
   A_3226_TSC01_AF.InpFaultAI := FALSE;
   A_3226_TSC01_AF.InpFaultDev := FALSE;
   A_3226_TSC01_AF.InHWStop := FALSE;
   A_3226_TSC01_AF.InDPFault := FALSE;
   A_3226_TSC01_AF.InDisable := FALSE;
   A_3226_TSC01_AF.CmdFaultReset := FALSE;
   A_3226_TSC01_AF.InLocal := FALSE;
   A_3226_TSC01_AF.spare0305 := FALSE;
   A_3226_TSC01_AF.InReport := FALSE;
   A_3226_TSC01_AF.spare0307 := FALSE;
   A_3226_TSC01_AF.OutLL := FALSE;
   A_3226_TSC01_AF.OutL := FALSE;
   A_3226_TSC01_AF.OutH := FALSE;
   A_3226_TSC01_AF.OutHH := FALSE;
   A_3226_TSC01_AF.OutOverflow := FALSE;
   A_3226_TSC01_AF.spare0405 := FALSE;
   A_3226_TSC01_AF.OutFaultAI := FALSE;
   A_3226_TSC01_AF.spare0407 := FALSE;
   A_3226_TSC01_AF.StLL := FALSE;
   A_3226_TSC01_AF.StL := FALSE;
   A_3226_TSC01_AF.StMid := FALSE;
   A_3226_TSC01_AF.StH := FALSE;
   A_3226_TSC01_AF.StHH := FALSE;
   A_3226_TSC01_AF.StFaultAI := FALSE;
   A_3226_TSC01_AF.OutWarning := FALSE;
   A_3226_TSC01_AF.OutFaulted := FALSE;
   A_3226_TSC01_AF.InpValue := 0;
   A_3226_TSC01_AF.OutValuePc := 0;
   A_3226_TSC01_AF.OutValueUnits := L#0;
   A_3226_TSC01_AF.Msg.WarningDoneLL := FALSE;
   A_3226_TSC01_AF.Msg.WarningDoneL := FALSE;
   A_3226_TSC01_AF.Msg.WarningDoneMid := FALSE;
   A_3226_TSC01_AF.Msg.WarningDoneH := FALSE;
   A_3226_TSC01_AF.Msg.WarningDoneHH := FALSE;
   A_3226_TSC01_AF.Msg.FaultDoneLL := FALSE;
   A_3226_TSC01_AF.Msg.FaultDoneL := FALSE;
   A_3226_TSC01_AF.Msg.FaultDoneMid := FALSE;
   A_3226_TSC01_AF.Msg.FaultDoneH := FALSE;
   A_3226_TSC01_AF.Msg.FaultDoneHH := FALSE;
   A_3226_TSC01_AF.Msg.FaultDoneDev := FALSE;
   A_3226_TSC01_AF.Msg.FaultDoneAI := FALSE;
   A_3226_TSC01_AF.OutAlarmNrLog := 0;
   A_3226_TSC01_AF.Par.ParObjectNo := 29724;
   A_3226_TSC01_AF.Par.ParMsgType := 7252;
   A_3226_TSC01_AF.Par.ParHornCode := 11;
   A_3226_TSC01_AF.Par.ParLogOff := FALSE;
   A_3226_TSC01_AF.Par.ParSpare0401 := FALSE;
   A_3226_TSC01_AF.Par.ParValueByUser := FALSE;
   A_3226_TSC01_AF.Par.ParLimitsPc := TRUE;
   A_3226_TSC01_AF.Par.ParWago := FALSE;
   A_3226_TSC01_AF.Par.ParNoHornByWarning := FALSE;
   A_3226_TSC01_AF.Par.ParWarningLL := FALSE;
   A_3226_TSC01_AF.Par.ParWarningL := FALSE;
   A_3226_TSC01_AF.Par.ParWarningMid := FALSE;
   A_3226_TSC01_AF.Par.ParWarningH := FALSE;
   A_3226_TSC01_AF.Par.ParWarningHH := FALSE;
   A_3226_TSC01_AF.Par.ParPreAlarmLL := FALSE;
   A_3226_TSC01_AF.Par.ParPreAlarmL := FALSE;
   A_3226_TSC01_AF.Par.ParPreAlarmMid := FALSE;
   A_3226_TSC01_AF.Par.ParPreAlarmH := FALSE;
   A_3226_TSC01_AF.Par.ParPreAlarmHH := FALSE;
   A_3226_TSC01_AF.Par.ParUnitsByZeroDigit := L#0;
   A_3226_TSC01_AF.Par.ParUnitsByMaxDigit := L#16880;
   A_3226_TSC01_AF.Par.ParUnitsBy100Pc := L#10000;
   A_3226_TSC01_AF.Par.ParLimitLL := L#-1;
   A_3226_TSC01_AF.Par.ParLimitL := L#3000;
   A_3226_TSC01_AF.Par.ParLimitH := L#10000;
   A_3226_TSC01_AF.Par.ParLimitHH := L#10100;
   A_3226_TSC01_AF.Par.ParMonTimeLL := 0;
   A_3226_TSC01_AF.Par.ParMonTimeL := 0;
   A_3226_TSC01_AF.Par.ParMonTimeMid := 0;
   A_3226_TSC01_AF.Par.ParMonTimeH := 0;
   A_3226_TSC01_AF.Par.ParMonTimeHH := 0;
   A_3226_TSC01_AF.Par.ParDelayTimeDown := 10;
   A_3226_TSC01_AF.Par.ParDelayTimeUp := 10;
   A_3226_TSC01_AF.Par.ParDelayTime := 30;
   A_3226_TSC01_AF.Par.OutMonTimeLL := 0;
   A_3226_TSC01_AF.Par.OutMonTimeL := 0;
   A_3226_TSC01_AF.Par.OutMonTimeMid := 0;
   A_3226_TSC01_AF.Par.OutMonTimeH := 0;
   A_3226_TSC01_AF.Par.OutMonTimeHH := 0;
   A_3226_TSC01_AF.Par.OutDelayTimeDown := 0;
   A_3226_TSC01_AF.Par.OutDelayTimeUp := 0;
   A_3226_TSC01_AF.Par.OutDelayTime := 0;
   A_3226_TSC01_AF.Par.Spare66 := 0;
   A_3226_TSC01_AP.StCode := 0;
   A_3226_TSC01_AP.InMonLL := FALSE;
   A_3226_TSC01_AP.InMonL := FALSE;
   A_3226_TSC01_AP.InMonMid := FALSE;
   A_3226_TSC01_AP.InMonH := FALSE;
   A_3226_TSC01_AP.InMonHH := FALSE;
   A_3226_TSC01_AP.spare0205 := FALSE;
   A_3226_TSC01_AP.InpFaultAI := FALSE;
   A_3226_TSC01_AP.InpFaultDev := FALSE;
   A_3226_TSC01_AP.InHWStop := FALSE;
   A_3226_TSC01_AP.InDPFault := FALSE;
   A_3226_TSC01_AP.InDisable := FALSE;
   A_3226_TSC01_AP.CmdFaultReset := FALSE;
   A_3226_TSC01_AP.InLocal := FALSE;
   A_3226_TSC01_AP.spare0305 := FALSE;
   A_3226_TSC01_AP.InReport := FALSE;
   A_3226_TSC01_AP.spare0307 := FALSE;
   A_3226_TSC01_AP.OutLL := FALSE;
   A_3226_TSC01_AP.OutL := FALSE;
   A_3226_TSC01_AP.OutH := FALSE;
   A_3226_TSC01_AP.OutHH := FALSE;
   A_3226_TSC01_AP.OutOverflow := FALSE;
   A_3226_TSC01_AP.spare0405 := FALSE;
   A_3226_TSC01_AP.OutFaultAI := FALSE;
   A_3226_TSC01_AP.spare0407 := FALSE;
   A_3226_TSC01_AP.StLL := FALSE;
   A_3226_TSC01_AP.StL := FALSE;
   A_3226_TSC01_AP.StMid := FALSE;
   A_3226_TSC01_AP.StH := FALSE;
   A_3226_TSC01_AP.StHH := FALSE;
   A_3226_TSC01_AP.StFaultAI := FALSE;
   A_3226_TSC01_AP.OutWarning := FALSE;
   A_3226_TSC01_AP.OutFaulted := FALSE;
   A_3226_TSC01_AP.InpValue := 0;
   A_3226_TSC01_AP.OutValuePc := 0;
   A_3226_TSC01_AP.OutValueUnits := L#0;
   A_3226_TSC01_AP.Msg.WarningDoneLL := FALSE;
   A_3226_TSC01_AP.Msg.WarningDoneL := FALSE;
   A_3226_TSC01_AP.Msg.WarningDoneMid := FALSE;
   A_3226_TSC01_AP.Msg.WarningDoneH := FALSE;
   A_3226_TSC01_AP.Msg.WarningDoneHH := FALSE;
   A_3226_TSC01_AP.Msg.FaultDoneLL := FALSE;
   A_3226_TSC01_AP.Msg.FaultDoneL := FALSE;
   A_3226_TSC01_AP.Msg.FaultDoneMid := FALSE;
   A_3226_TSC01_AP.Msg.FaultDoneH := FALSE;
   A_3226_TSC01_AP.Msg.FaultDoneHH := FALSE;
   A_3226_TSC01_AP.Msg.FaultDoneDev := FALSE;
   A_3226_TSC01_AP.Msg.FaultDoneAI := FALSE;
   A_3226_TSC01_AP.OutAlarmNrLog := 0;
   A_3226_TSC01_AP.Par.ParObjectNo := 29725;
   A_3226_TSC01_AP.Par.ParMsgType := 7252;
   A_3226_TSC01_AP.Par.ParHornCode := 11;
   A_3226_TSC01_AP.Par.ParLogOff := FALSE;
   A_3226_TSC01_AP.Par.ParSpare0401 := FALSE;
   A_3226_TSC01_AP.Par.ParValueByUser := FALSE;
   A_3226_TSC01_AP.Par.ParLimitsPc := TRUE;
   A_3226_TSC01_AP.Par.ParWago := FALSE;
   A_3226_TSC01_AP.Par.ParNoHornByWarning := FALSE;
   A_3226_TSC01_AP.Par.ParWarningLL := FALSE;
   A_3226_TSC01_AP.Par.ParWarningL := FALSE;
   A_3226_TSC01_AP.Par.ParWarningMid := FALSE;
   A_3226_TSC01_AP.Par.ParWarningH := FALSE;
   A_3226_TSC01_AP.Par.ParWarningHH := FALSE;
   A_3226_TSC01_AP.Par.ParPreAlarmLL := FALSE;
   A_3226_TSC01_AP.Par.ParPreAlarmL := FALSE;
   A_3226_TSC01_AP.Par.ParPreAlarmMid := FALSE;
   A_3226_TSC01_AP.Par.ParPreAlarmH := FALSE;
   A_3226_TSC01_AP.Par.ParPreAlarmHH := FALSE;
   A_3226_TSC01_AP.Par.ParUnitsByZeroDigit := L#0;
   A_3226_TSC01_AP.Par.ParUnitsByMaxDigit := L#16384;
   A_3226_TSC01_AP.Par.ParUnitsBy100Pc := L#10000;
   A_3226_TSC01_AP.Par.ParLimitLL := L#-1;
   A_3226_TSC01_AP.Par.ParLimitL := L#0;
   A_3226_TSC01_AP.Par.ParLimitH := L#3150;
   A_3226_TSC01_AP.Par.ParLimitHH := L#3500;
   A_3226_TSC01_AP.Par.ParMonTimeLL := 0;
   A_3226_TSC01_AP.Par.ParMonTimeL := 0;
   A_3226_TSC01_AP.Par.ParMonTimeMid := 0;
   A_3226_TSC01_AP.Par.ParMonTimeH := 0;
   A_3226_TSC01_AP.Par.ParMonTimeHH := 0;
   A_3226_TSC01_AP.Par.ParDelayTimeDown := 10;
   A_3226_TSC01_AP.Par.ParDelayTimeUp := 10;
   A_3226_TSC01_AP.Par.ParDelayTime := 30;
   A_3226_TSC01_AP.Par.OutMonTimeLL := 0;
   A_3226_TSC01_AP.Par.OutMonTimeL := 0;
   A_3226_TSC01_AP.Par.OutMonTimeMid := 0;
   A_3226_TSC01_AP.Par.OutMonTimeH := 0;
   A_3226_TSC01_AP.Par.OutMonTimeHH := 0;
   A_3226_TSC01_AP.Par.OutDelayTimeDown := 0;
   A_3226_TSC01_AP.Par.OutDelayTimeUp := 0;
   A_3226_TSC01_AP.Par.OutDelayTime := 0;
   A_3226_TSC01_AP.Par.Spare66 := 0;
   A_3226_TSC01_AT.StCode := 0;
   A_3226_TSC01_AT.InMonLL := FALSE;
   A_3226_TSC01_AT.InMonL := FALSE;
   A_3226_TSC01_AT.InMonMid := FALSE;
   A_3226_TSC01_AT.InMonH := FALSE;
   A_3226_TSC01_AT.InMonHH := FALSE;
   A_3226_TSC01_AT.spare0205 := FALSE;
   A_3226_TSC01_AT.InpFaultAI := FALSE;
   A_3226_TSC01_AT.InpFaultDev := FALSE;
   A_3226_TSC01_AT.InHWStop := FALSE;
   A_3226_TSC01_AT.InDPFault := FALSE;
   A_3226_TSC01_AT.InDisable := FALSE;
   A_3226_TSC01_AT.CmdFaultReset := FALSE;
   A_3226_TSC01_AT.InLocal := FALSE;
   A_3226_TSC01_AT.spare0305 := FALSE;
   A_3226_TSC01_AT.InReport := FALSE;
   A_3226_TSC01_AT.spare0307 := FALSE;
   A_3226_TSC01_AT.OutLL := FALSE;
   A_3226_TSC01_AT.OutL := FALSE;
   A_3226_TSC01_AT.OutH := FALSE;
   A_3226_TSC01_AT.OutHH := FALSE;
   A_3226_TSC01_AT.OutOverflow := FALSE;
   A_3226_TSC01_AT.spare0405 := FALSE;
   A_3226_TSC01_AT.OutFaultAI := FALSE;
   A_3226_TSC01_AT.spare0407 := FALSE;
   A_3226_TSC01_AT.StLL := FALSE;
   A_3226_TSC01_AT.StL := FALSE;
   A_3226_TSC01_AT.StMid := FALSE;
   A_3226_TSC01_AT.StH := FALSE;
   A_3226_TSC01_AT.StHH := FALSE;
   A_3226_TSC01_AT.StFaultAI := FALSE;
   A_3226_TSC01_AT.OutWarning := FALSE;
   A_3226_TSC01_AT.OutFaulted := FALSE;
   A_3226_TSC01_AT.InpValue := 0;
   A_3226_TSC01_AT.OutValuePc := 0;
   A_3226_TSC01_AT.OutValueUnits := L#0;
   A_3226_TSC01_AT.Msg.WarningDoneLL := FALSE;
   A_3226_TSC01_AT.Msg.WarningDoneL := FALSE;
   A_3226_TSC01_AT.Msg.WarningDoneMid := FALSE;
   A_3226_TSC01_AT.Msg.WarningDoneH := FALSE;
   A_3226_TSC01_AT.Msg.WarningDoneHH := FALSE;
   A_3226_TSC01_AT.Msg.FaultDoneLL := FALSE;
   A_3226_TSC01_AT.Msg.FaultDoneL := FALSE;
   A_3226_TSC01_AT.Msg.FaultDoneMid := FALSE;
   A_3226_TSC01_AT.Msg.FaultDoneH := FALSE;
   A_3226_TSC01_AT.Msg.FaultDoneHH := FALSE;
   A_3226_TSC01_AT.Msg.FaultDoneDev := FALSE;
   A_3226_TSC01_AT.Msg.FaultDoneAI := FALSE;
   A_3226_TSC01_AT.OutAlarmNrLog := 0;
   A_3226_TSC01_AT.Par.ParObjectNo := 29726;
   A_3226_TSC01_AT.Par.ParMsgType := 7252;
   A_3226_TSC01_AT.Par.ParHornCode := 11;
   A_3226_TSC01_AT.Par.ParLogOff := FALSE;
   A_3226_TSC01_AT.Par.ParSpare0401 := FALSE;
   A_3226_TSC01_AT.Par.ParValueByUser := FALSE;
   A_3226_TSC01_AT.Par.ParLimitsPc := TRUE;
   A_3226_TSC01_AT.Par.ParWago := FALSE;
   A_3226_TSC01_AT.Par.ParNoHornByWarning := FALSE;
   A_3226_TSC01_AT.Par.ParWarningLL := FALSE;
   A_3226_TSC01_AT.Par.ParWarningL := FALSE;
   A_3226_TSC01_AT.Par.ParWarningMid := FALSE;
   A_3226_TSC01_AT.Par.ParWarningH := FALSE;
   A_3226_TSC01_AT.Par.ParWarningHH := FALSE;
   A_3226_TSC01_AT.Par.ParPreAlarmLL := FALSE;
   A_3226_TSC01_AT.Par.ParPreAlarmL := FALSE;
   A_3226_TSC01_AT.Par.ParPreAlarmMid := FALSE;
   A_3226_TSC01_AT.Par.ParPreAlarmH := FALSE;
   A_3226_TSC01_AT.Par.ParPreAlarmHH := FALSE;
   A_3226_TSC01_AT.Par.ParUnitsByZeroDigit := L#0;
   A_3226_TSC01_AT.Par.ParUnitsByMaxDigit := L#16384;
   A_3226_TSC01_AT.Par.ParUnitsBy100Pc := L#10000;
   A_3226_TSC01_AT.Par.ParLimitLL := L#-1;
   A_3226_TSC01_AT.Par.ParLimitL := L#0;
   A_3226_TSC01_AT.Par.ParLimitH := L#7000;
   A_3226_TSC01_AT.Par.ParLimitHH := L#8000;
   A_3226_TSC01_AT.Par.ParMonTimeLL := 0;
   A_3226_TSC01_AT.Par.ParMonTimeL := 0;
   A_3226_TSC01_AT.Par.ParMonTimeMid := 0;
   A_3226_TSC01_AT.Par.ParMonTimeH := 0;
   A_3226_TSC01_AT.Par.ParMonTimeHH := 0;
   A_3226_TSC01_AT.Par.ParDelayTimeDown := 10;
   A_3226_TSC01_AT.Par.ParDelayTimeUp := 10;
   A_3226_TSC01_AT.Par.ParDelayTime := 30;
   A_3226_TSC01_AT.Par.OutMonTimeLL := 0;
   A_3226_TSC01_AT.Par.OutMonTimeL := 0;
   A_3226_TSC01_AT.Par.OutMonTimeMid := 0;
   A_3226_TSC01_AT.Par.OutMonTimeH := 0;
   A_3226_TSC01_AT.Par.OutMonTimeHH := 0;
   A_3226_TSC01_AT.Par.OutDelayTimeDown := 0;
   A_3226_TSC01_AT.Par.OutDelayTimeUp := 0;
   A_3226_TSC01_AT.Par.OutDelayTime := 0;
   A_3226_TSC01_AT.Par.Spare66 := 0;
   A_3226_TSC01_COM.InValuePC := 0;
   A_3226_TSC01_COM.InEnableRev := FALSE;
   A_3226_TSC01_COM.InEnableFwd := FALSE;
   A_3226_TSC01_COM.CmdFaultReset := FALSE;
   A_3226_TSC01_COM.OutRunningRev := FALSE;
   A_3226_TSC01_COM.OutRunningFwd := FALSE;
   A_3226_TSC01_COM.OutFault := FALSE;
   A_3226_TSC01_COM.MotorStStopped := FALSE;
   A_3226_TSC01_COM.Spare := FALSE;
   A_3226_TSC01_COM.OutValuePC := 0;
   A_3226_TSC01_COM.Input.StateWord_1.STATE_WORD_BIT_8 := FALSE;
   A_3226_TSC01_COM.Input.StateWord_1.STATE_WORD_BIT_9 := FALSE;
   A_3226_TSC01_COM.Input.StateWord_1.STATE_WORD_BIT_10 := FALSE;
   A_3226_TSC01_COM.Input.StateWord_1.STATE_WORD_BIT_11 := FALSE;
   A_3226_TSC01_COM.Input.StateWord_1.STATE_WORD_BIT_12 := FALSE;
   A_3226_TSC01_COM.Input.StateWord_1.STATE_WORD_BIT_13 := FALSE;
   A_3226_TSC01_COM.Input.StateWord_1.STATE_WORD_BIT_14 := FALSE;
   A_3226_TSC01_COM.Input.StateWord_1.STATE_WORD_BIT_15 := FALSE;
   A_3226_TSC01_COM.Input.StateWord_1.ENDSTUFE_FREIGEGEBEN := FALSE;
   A_3226_TSC01_COM.Input.StateWord_1.BETRIEBSBEREIT := FALSE;
   A_3226_TSC01_COM.Input.StateWord_1.PA_DATEN_FREIGEGEBEN := FALSE;
   A_3226_TSC01_COM.Input.StateWord_1.AKTUELL_INTEGRATORSATZ := FALSE;
   A_3226_TSC01_COM.Input.StateWord_1.AKTUELL_PARAMETERSATZ := FALSE;
   A_3226_TSC01_COM.Input.StateWord_1.STOERUNG_WARNUNG := FALSE;
   A_3226_TSC01_COM.Input.StateWord_1.LS_RECHTS_AKTIV := FALSE;
   A_3226_TSC01_COM.Input.StateWord_1.LS_LINKS_AKTIV := FALSE;
   A_3226_TSC01_COM.Input.ActualValue01 := 0;
   A_3226_TSC01_COM.Input.ActualValue02 := 0;
   A_3226_TSC01_COM.Input.ActualValue03 := 0;
   A_3226_TSC01_COM.Input.ActualValue04 := 0;
   A_3226_TSC01_COM.Input.ActualValue05 := 0;
   A_3226_TSC01_COM.Output.ControlWord_1.CONTROL_WORD_BIT_8 := FALSE;
   A_3226_TSC01_COM.Output.ControlWord_1.CONTROL_WORD_BIT_9 := FALSE;
   A_3226_TSC01_COM.Output.ControlWord_1.CONTROL_WORD_BIT_10 := FALSE;
   A_3226_TSC01_COM.Output.ControlWord_1.CONTROL_WORD_BIT_11 := FALSE;
   A_3226_TSC01_COM.Output.ControlWord_1.CONTROL_WORD_BIT_12 := FALSE;
   A_3226_TSC01_COM.Output.ControlWord_1.CONTROL_WORD_BIT_13 := FALSE;
   A_3226_TSC01_COM.Output.ControlWord_1.CONTROL_WORD_BIT_14 := FALSE;
   A_3226_TSC01_COM.Output.ControlWord_1.CONTROL_WORD_BIT_15 := FALSE;
   A_3226_TSC01_COM.Output.ControlWord_1.REGLERSPERRE := FALSE;
   A_3226_TSC01_COM.Output.ControlWord_1.FREIGABE_SCHNELLSTOPP := FALSE;
   A_3226_TSC01_COM.Output.ControlWord_1.FREIGABE_HALT := FALSE;
   A_3226_TSC01_COM.Output.ControlWord_1.HALTEREGELUNG := FALSE;
   A_3226_TSC01_COM.Output.ControlWord_1.INTEGRATOR := FALSE;
   A_3226_TSC01_COM.Output.ControlWord_1.PARAMETERSATZ := FALSE;
   A_3226_TSC01_COM.Output.ControlWord_1.RESET := FALSE;
   A_3226_TSC01_COM.Output.ControlWord_1.RESERVE_BIT_7 := FALSE;
   A_3226_TSC01_COM.Output.SetpointValue01 := 0;
   A_3226_TSC01_COM.Output.SetpointValue02 := 0;
   A_3226_TSC01_COM.Output.SetpointValue03 := 0;
   A_3226_TSC01_COM.Output.SetpointValue04 := 0;
   A_3226_TSC01_COM.Output.SetpointValue05 := 0;
   A_3226_TSC01_COM.Par.spare1 := 0;
   A_3226_TSC01_COM.Par.spare2 := 0;
   A_3226_TSC01_COM.Par.spare3 := 0;
   A_3226_TSC01_COM.Par.ParMovidrive := TRUE;
   A_3226_TSC01_COM.Par.ParSinamics := FALSE;
   A_3226_TSC01_COM.Par.ParMicromaster := FALSE;
   A_3226_TSC01_COM.Par.ParABB := FALSE;
   A_3226_TSC01_COM.Par.ParNord := FALSE;
   A_3226_TSC01_COM.Par.ParDanfoss := FALSE;
   A_3226_TSC01_COM.Par.ParIOByteNo := 0;
      #A_3225_TSC01_COM.Par.ParMovidrive                            :=1;
      #A_3225_TSC01_COM.Par.ParSinamics                             :=0;
      #A_3225_TSC01_COM.Par.ParMicromaster                          :=0;
      #A_3225_TSC01_COM.Par.ParABB                                  :=0;
      #A_3225_TSC01_COM.Par.ParNord                                 :=0;
      #A_3225_TSC01_COM.Par.ParDanfoss                              :=0;
      #A_3225_TSC01_COM.Par.ParIOByteNo                             :=0;
      #A_3225_TSC01_AC.Par.ParObjectNo                             :=29710;
      #A_3225_TSC01_AC.Par.ParHornCode                             :=11;
      #A_3225_TSC01_AC.Par.ParMsgType                              :=7252;
      #A_3225_TSC01_AC.Par.ParUnitsByZeroDigit                     :=L#0;
      #A_3225_TSC01_AC.Par.ParUnitsByMaxDigit                      :=L#25384;
      #A_3225_TSC01_AC.Par.ParUnitsBy100Pc                         :=L#10000;
      #A_3225_TSC01_AC.Par.ParDelayTimeDown                        :=10;
      #A_3225_TSC01_AC.Par.ParDelayTimeUp                          :=10;
      #A_3225_TSC01_AC.Par.ParDelayTime                            :=30;
      #A_3225_TSC01_AC.Par.ParLimitLL                              :=L#-1;
      #A_3225_TSC01_AC.Par.ParLimitL                               :=L#0;
      #A_3225_TSC01_AC.Par.ParLimitH                               :=L#5400;
      #A_3225_TSC01_AC.Par.ParLimitHH                              :=L#6000;
      #A_3225_TSC01_AC.Par.ParMonTimeLL                            :=0;
      #A_3225_TSC01_AC.Par.ParMonTimeL                             :=0;
      #A_3225_TSC01_AC.Par.ParMonTimeMid                           :=0;
      #A_3225_TSC01_AC.Par.ParMonTimeH                             :=0;
      #A_3225_TSC01_AC.Par.ParMonTimeHH                            :=0;
      #A_3225_TSC01_AC.Par.ParLogOff                               :=False;
      #A_3225_TSC01_AC.Par.ParValueByUser                          :=False;
      #A_3225_TSC01_AC.Par.ParLimitsPc                             :=True;
      #A_3225_TSC01_AC.Par.ParWago                                 :=False;
      #A_3225_TSC01_AC.Par.ParNoHornByWarning                      :=False;
      #A_3225_TSC01_AC.Par.ParWarningLL                            :=False;
      #A_3225_TSC01_AC.Par.ParWarningL                             :=False;
      #A_3225_TSC01_AC.Par.ParWarningMid                           :=False;
      #A_3225_TSC01_AC.Par.ParWarningH                             :=False;
      #A_3225_TSC01_AC.Par.ParWarningHH                            :=False;
      #A_3225_TSC01_AC.Par.ParPreAlarmLL                           :=False;
      #A_3225_TSC01_AC.Par.ParPreAlarmL                            :=False;
      #A_3225_TSC01_AC.Par.ParPreAlarmMid                          :=False;
      #A_3225_TSC01_AC.Par.ParPreAlarmH                            :=False;
      #A_3225_TSC01_AC.Par.ParPreAlarmHH                           :=False;
      #A_3225_TSC01_AF.Par.ParObjectNo                             :=29711;
      #A_3225_TSC01_AF.Par.ParHornCode                             :=11;
      #A_3225_TSC01_AF.Par.ParMsgType                              :=7252;
      #A_3225_TSC01_AF.Par.ParUnitsByZeroDigit                     :=L#0;
      #A_3225_TSC01_AF.Par.ParUnitsByMaxDigit                      :=L#16880;
      #A_3225_TSC01_AF.Par.ParUnitsBy100Pc                         :=L#10000;
      #A_3225_TSC01_AF.Par.ParDelayTimeDown                        :=10;
      #A_3225_TSC01_AF.Par.ParDelayTimeUp                          :=10;
      #A_3225_TSC01_AF.Par.ParDelayTime                            :=30;
      #A_3225_TSC01_AF.Par.ParLimitLL                              :=L#-1;
      #A_3225_TSC01_AF.Par.ParLimitL                               :=L#3000;
      #A_3225_TSC01_AF.Par.ParLimitH                               :=L#10000;
      #A_3225_TSC01_AF.Par.ParLimitHH                              :=L#10100;
      #A_3225_TSC01_AF.Par.ParMonTimeLL                            :=0;
      #A_3225_TSC01_AF.Par.ParMonTimeL                             :=0;
      #A_3225_TSC01_AF.Par.ParMonTimeMid                           :=0;
      #A_3225_TSC01_AF.Par.ParMonTimeH                             :=0;
      #A_3225_TSC01_AF.Par.ParMonTimeHH                            :=0;
      #A_3225_TSC01_AF.Par.ParLogOff                               :=False;
      #A_3225_TSC01_AF.Par.ParValueByUser                          :=False;
      #A_3225_TSC01_AF.Par.ParLimitsPc                             :=True;
      #A_3225_TSC01_AF.Par.ParWago                                 :=False;
      #A_3225_TSC01_AF.Par.ParNoHornByWarning                      :=False;
      #A_3225_TSC01_AF.Par.ParWarningLL                            :=False;
      #A_3225_TSC01_AF.Par.ParWarningL                             :=False;
      #A_3225_TSC01_AF.Par.ParWarningMid                           :=False;
      #A_3225_TSC01_AF.Par.ParWarningH                             :=False;
      #A_3225_TSC01_AF.Par.ParWarningHH                            :=False;
      #A_3225_TSC01_AF.Par.ParPreAlarmLL                           :=False;
      #A_3225_TSC01_AF.Par.ParPreAlarmL                            :=False;
      #A_3225_TSC01_AF.Par.ParPreAlarmMid                          :=False;
      #A_3225_TSC01_AF.Par.ParPreAlarmH                            :=False;
      #A_3225_TSC01_AF.Par.ParPreAlarmHH                           :=False;
      #A_3225_TSC01_AP.Par.ParObjectNo                             :=29712;
      #A_3225_TSC01_AP.Par.ParHornCode                             :=11;
      #A_3225_TSC01_AP.Par.ParMsgType                              :=7252;
      #A_3225_TSC01_AP.Par.ParUnitsByZeroDigit                     :=L#0;
      #A_3225_TSC01_AP.Par.ParUnitsByMaxDigit                      :=L#16384;
      #A_3225_TSC01_AP.Par.ParUnitsBy100Pc                         :=L#10000;
      #A_3225_TSC01_AP.Par.ParDelayTimeDown                        :=10;
      #A_3225_TSC01_AP.Par.ParDelayTimeUp                          :=10;
      #A_3225_TSC01_AP.Par.ParDelayTime                            :=30;
      #A_3225_TSC01_AP.Par.ParLimitLL                              :=L#-1;
      #A_3225_TSC01_AP.Par.ParLimitL                               :=L#0;
      #A_3225_TSC01_AP.Par.ParLimitH                               :=L#3150;
      #A_3225_TSC01_AP.Par.ParLimitHH                              :=L#3500;
      #A_3225_TSC01_AP.Par.ParMonTimeLL                            :=0;
      #A_3225_TSC01_AP.Par.ParMonTimeL                             :=0;
      #A_3225_TSC01_AP.Par.ParMonTimeMid                           :=0;
      #A_3225_TSC01_AP.Par.ParMonTimeH                             :=0;
      #A_3225_TSC01_AP.Par.ParMonTimeHH                            :=0;
      #A_3225_TSC01_AP.Par.ParLogOff                               :=False;
      #A_3225_TSC01_AP.Par.ParValueByUser                          :=False;
      #A_3225_TSC01_AP.Par.ParLimitsPc                             :=True;
      #A_3225_TSC01_AP.Par.ParWago                                 :=False;
      #A_3225_TSC01_AP.Par.ParNoHornByWarning                      :=False;
      #A_3225_TSC01_AP.Par.ParWarningLL                            :=False;
      #A_3225_TSC01_AP.Par.ParWarningL                             :=False;
      #A_3225_TSC01_AP.Par.ParWarningMid                           :=False;
      #A_3225_TSC01_AP.Par.ParWarningH                             :=False;
      #A_3225_TSC01_AP.Par.ParWarningHH                            :=False;
      #A_3225_TSC01_AP.Par.ParPreAlarmLL                           :=False;
      #A_3225_TSC01_AP.Par.ParPreAlarmL                            :=False;
      #A_3225_TSC01_AP.Par.ParPreAlarmMid                          :=False;
      #A_3225_TSC01_AP.Par.ParPreAlarmH                            :=False;
      #A_3225_TSC01_AP.Par.ParPreAlarmHH                           :=False;
      #A_3225_TSC01_AT.Par.ParObjectNo                             :=29713;
      #A_3225_TSC01_AT.Par.ParHornCode                             :=11;
      #A_3225_TSC01_AT.Par.ParMsgType                              :=7252;
      #A_3225_TSC01_AT.Par.ParUnitsByZeroDigit                     :=L#0;
      #A_3225_TSC01_AT.Par.ParUnitsByMaxDigit                      :=L#16384;
      #A_3225_TSC01_AT.Par.ParUnitsBy100Pc                         :=L#10000;
      #A_3225_TSC01_AT.Par.ParDelayTimeDown                        :=10;
      #A_3225_TSC01_AT.Par.ParDelayTimeUp                          :=10;
      #A_3225_TSC01_AT.Par.ParDelayTime                            :=30;
      #A_3225_TSC01_AT.Par.ParLimitLL                              :=L#-1;
      #A_3225_TSC01_AT.Par.ParLimitL                               :=L#0;
      #A_3225_TSC01_AT.Par.ParLimitH                               :=L#7000;
      #A_3225_TSC01_AT.Par.ParLimitHH                              :=L#8000;
      #A_3225_TSC01_AT.Par.ParMonTimeLL                            :=0;
      #A_3225_TSC01_AT.Par.ParMonTimeL                             :=0;
      #A_3225_TSC01_AT.Par.ParMonTimeMid                           :=0;
      #A_3225_TSC01_AT.Par.ParMonTimeH                             :=0;
      #A_3225_TSC01_AT.Par.ParMonTimeHH                            :=0;
      #A_3225_TSC01_AT.Par.ParLogOff                               :=False;
      #A_3225_TSC01_AT.Par.ParValueByUser                          :=False;
      #A_3225_TSC01_AT.Par.ParLimitsPc                             :=True;
      #A_3225_TSC01_AT.Par.ParWago                                 :=False;
      #A_3225_TSC01_AT.Par.ParNoHornByWarning                      :=False;
      #A_3225_TSC01_AT.Par.ParWarningLL                            :=False;
      #A_3225_TSC01_AT.Par.ParWarningL                             :=False;
      #A_3225_TSC01_AT.Par.ParWarningMid                           :=False;
      #A_3225_TSC01_AT.Par.ParWarningH                             :=False;
      #A_3225_TSC01_AT.Par.ParWarningHH                            :=False;
      #A_3225_TSC01_AT.Par.ParPreAlarmLL                           :=False;
      #A_3225_TSC01_AT.Par.ParPreAlarmL                            :=False;
      #A_3225_TSC01_AT.Par.ParPreAlarmMid                          :=False;
      #A_3225_TSC01_AT.Par.ParPreAlarmH                            :=False;
      #A_3225_TSC01_AT.Par.ParPreAlarmHH                           :=False;
      #A_3225_TSC01.Par.ParObjectNo                             :=29705;
      #A_3225_TSC01.Par.ParMsgType                              :=7156;
      #A_3225_TSC01.Par.ParHornCode                             :=0;
      #A_3225_TSC01.Par.ParDelayChange                          :=20;
      #A_3225_TSC01.Par.ParDelayTrue                            :=10;
      #A_3225_TSC01.Par.ParDelayFalse                           :=0;
      #A_3225_TSC01.Par.ParTimeoutTrue                          :=0;
      #A_3225_TSC01.Par.ParTimeoutFalse                         :=0;
      #A_3225_TSC01.Par.ParLogOff                               :=False;
      #A_3225_TSC01.Par.Par2WorkingCond                         :=False;
      #A_3225_TSC01.Par.ParFaultRetry                           :=False;
      #A_3225_TSC01.Par.ParBinLevel                             :=False;
END_DATA_BLOCK

